(* IEC 61131-3 sources: RL_MAR/experiments/results/ablation/Ablation_no_post_process_deepseek-ai_DeepSeek-V3.2_20260602_235132 (part 2) *)

(* ---- med_34.st ---- *)
(*
    Coffee Machine Control Function Block
    Implements sequential control for water heating, grinding, and brewing
    Only one process active at a time
    Resets when start button is released
*)

FUNCTION_BLOCK CoffeeMachineControl
VAR_INPUT
    StartButton : BOOL;                    (* Start/run command *)
    ElapsedTime : DINT;                    (* Time elapsed since process start in ms *)
END_VAR

VAR_OUTPUT
    WaterHeating : BOOL;                   (* Control signal for water heater *)
    GrinderRunning : BOOL;                 (* Control signal for coffee grinder *)
    Brewing : BOOL;                        (* Control signal for brewing pump *)
    WaterHeated : BOOL;                    (* Status: Water heating complete *)
    GrinderFinished : BOOL;                (* Status: Grinding complete *)
    CoffeeReady : BOOL;                    (* Status: Brewing complete *)
END_VAR

VAR
    (* Process timing constants *)
    WaterHeatingDuration : DINT := 30000;  (* 30 seconds in milliseconds *)
    GrinderDuration : DINT := 15000;       (* 15 seconds in milliseconds *)
    BrewingDuration : DINT := 60000;       (* 60 seconds in milliseconds *)

    (* State management *)
    CurrentState : INT := 0;               (* 0=Idle, 1=Heating, 2=Grinding, 3=Brewing *)
    StateStartTime : DINT := 0;            (* Time when current state started *)
    PreviousStartButton : BOOL := FALSE;   (* Edge detection for start button *)

    (* Internal flags *)
    InternalWaterHeated : BOOL := FALSE;
    InternalGrinderFinished : BOOL := FALSE;
    InternalCoffeeReady : BOOL := FALSE;
END_VAR

(* Main control logic *)
IF NOT StartButton THEN
    (* Reset all outputs and state when start button is not pressed *)
    CurrentState := 0;
    StateStartTime := 0;
    WaterHeating := FALSE;
    GrinderRunning := FALSE;
    Brewing := FALSE;
    InternalWaterHeated := FALSE;
    InternalGrinderFinished := FALSE;
    InternalCoffeeReady := FALSE;
ELSE
    (* Detect rising edge of start button *)
    IF StartButton AND NOT PreviousStartButton AND CurrentState = 0 THEN
        (* Start new cycle from idle state *)
        CurrentState := 1;
        StateStartTime := ElapsedTime;
        InternalWaterHeated := FALSE;
        InternalGrinderFinished := FALSE;
        InternalCoffeeReady := FALSE;
    END_IF;

    (* State machine execution *)
    CASE CurrentState OF
        0: (* Idle State *)
            WaterHeating := FALSE;
            GrinderRunning := FALSE;
            Brewing := FALSE;

        1: (* Water Heating State *)
            WaterHeating := TRUE;
            GrinderRunning := FALSE;
            Brewing := FALSE;

            (* Check if heating duration completed *)
            IF (ElapsedTime - StateStartTime) >= WaterHeatingDuration THEN
                InternalWaterHeated := TRUE;
                WaterHeating := FALSE;
                CurrentState := 2;
                StateStartTime := ElapsedTime;
            END_IF;

        2: (* Grinding State *)
            WaterHeating := FALSE;
            GrinderRunning := TRUE;
            Brewing := FALSE;

            (* Check if grinding duration completed *)
            IF (ElapsedTime - StateStartTime) >= GrinderDuration THEN
                InternalGrinderFinished := TRUE;
                GrinderRunning := FALSE;
                CurrentState := 3;
                StateStartTime := ElapsedTime;
            END_IF;

        3: (* Brewing State *)
            WaterHeating := FALSE;
            GrinderRunning := FALSE;
            Brewing := TRUE;

            (* Check if brewing duration completed *)
            IF (ElapsedTime - StateStartTime) >= BrewingDuration THEN
                InternalCoffeeReady := TRUE;
                Brewing := FALSE;
                CurrentState := 0;  (* Return to idle after completion *)
            END_IF;
    END_CASE;
END_IF;

(* Update status outputs *)
WaterHeated := InternalWaterHeated;
GrinderFinished := InternalGrinderFinished;
CoffeeReady := InternalCoffeeReady;

(* Store previous start button state for edge detection *)
PreviousStartButton := StartButton;

END_FUNCTION_BLOCK;

(* ---- med_35.st ---- *)
FUNCTION_BLOCK FB_SimpleCalculation
VAR_INPUT
    INPUT_VAR1 : INT := 2;
    VAR2 : INT := 0;
END_VAR

VAR_OUTPUT
    OUTPUT_VAR1 : INT;
    OUTPUT_VAR2 : INT;
END_VAR

VAR
    i : INT; // Loop counter for multiplication loop
    COUNTER2 : INT := 0;
END_VAR

// Initialize outputs from inputs
OUTPUT_VAR1 := INPUT_VAR1;
OUTPUT_VAR2 := VAR2;

// First loop: Multiply OUTPUT_VAR1 by 2 for exactly 5 iterations
FOR i := 1 TO 5 DO
    OUTPUT_VAR1 := OUTPUT_VAR1 * 2;
END_FOR;

// Second loop: Increment OUTPUT_VAR2 by 1 for exactly 5 iterations
COUNTER2 := 0;
WHILE COUNTER2 < 5 DO
    OUTPUT_VAR2 := OUTPUT_VAR2 + 1;
    COUNTER2 := COUNTER2 + 1;
END_WHILE;

END_FUNCTION_BLOCK

(* ---- med_36.st ---- *)
TYPE
    Point2D : STRUCT
        X : INT;
        Y : INT;
    END_STRUCT;
END_TYPE

FUNCTION_BLOCK FB_ExpandedPoint
    VAR_INPUT
        INPUT_VAR2 : INT;
        INPUT_VAR1_X : INT;
        INPUT_VAR1_Y : INT;
        INPUT_VAR3_X : INT := 1;
        INPUT_VAR3_Y : INT := 2;
    END_VAR

    VAR_OUTPUT
        OUTPUT_VAR2 : INT;
        OUTPUT_VAR1_X : INT;
        OUTPUT_VAR1_Y : INT;
        OUTPUT_VAR3_X : INT;
        OUTPUT_VAR3_Y : INT;
    END_VAR

    VAR
        // Internal structured variables for cleaner code organization
        Internal_INPUT_VAR1 : Point2D;
        Internal_INPUT_VAR3 : Point2D;
        Internal_OUTPUT_VAR1 : Point2D;
        Internal_OUTPUT_VAR3 : Point2D;
    END_VAR

    // Main execution logic
    OUTPUT_VAR2 := INPUT_VAR2;

    // Set OUTPUT_VAR1_X and OUTPUT_VAR1_Y to fixed constants as specified
    OUTPUT_VAR1_X := 1;
    OUTPUT_VAR1_Y := 2;

    // Set OUTPUT_VAR3_X and OUTPUT_VAR3_Y to fixed constants as specified
    OUTPUT_VAR3_X := 100;
    OUTPUT_VAR3_Y := -7000;

    // Optional: Update internal structured variables for consistency
    Internal_OUTPUT_VAR1.X := OUTPUT_VAR1_X;
    Internal_OUTPUT_VAR1.Y := OUTPUT_VAR1_Y;
    Internal_OUTPUT_VAR3.X := OUTPUT_VAR3_X;
    Internal_OUTPUT_VAR3.Y := OUTPUT_VAR3_Y;

    // Store input values in internal structured variables (for potential future use)
    Internal_INPUT_VAR1.X := INPUT_VAR1_X;
    Internal_INPUT_VAR1.Y := INPUT_VAR1_Y;
    Internal_INPUT_VAR3.X := INPUT_VAR3_X;
    Internal_INPUT_VAR3.Y := INPUT_VAR3_Y;

END_FUNCTION_BLOCK

(* ---- med_37.st ---- *)
FUNCTION_BLOCK FB_RealValueAdjuster
VAR_INPUT
    x_in : REAL;
END_VAR

VAR_OUTPUT
    x_out : REAL;
END_VAR

VAR
    x_int : INT;
END_VAR

x_out := x_in;

IF x_in = 0.0 THEN
    x_out := x_out + 1.0;
END_IF;

IF x_in <> 0.0 THEN
    x_out := x_out + 1.0;
END_IF;

x_int := REAL_TO_INT(x_in);
IF x_int <> 0 THEN
    x_out := x_out + 1.0;
END_IF;

END_FUNCTION_BLOCK

(* ---- med_38.st ---- *)
FUNCTION_BLOCK SolarPanelTracking
VAR_INPUT
    SolarIntensity : REAL;      (* Input: Solar intensity in percentage *)
    CurrentTime : TIME;         (* Input: Current time of day *)
END_VAR

VAR_OUTPUT
    PanelAngle : REAL := 0.0;   (* Output: Panel angle in degrees *)
END_VAR

VAR
    SunriseTime : TIME := T#6H;    (* Sunrise time set to 6 AM *)
    SunsetTime : TIME := T#18H;    (* Sunset time set to 6 PM *)
    NoonTime : TIME := T#12H;      (* Noon time set to 12 PM *)
    MorningAngle : REAL := 30.0;   (* Angle during morning *)
    NoonAngle : REAL := 60.0;      (* Angle during noon *)
    EveningAngle : REAL := 30.0;   (* Angle during evening *)
    State : INT := 0;              (* Current state *)
    NextState : INT := 0;          (* Next state *)
END_VAR

(* State machine implementation *)
CASE State OF
    0: (* INIT *)
        PanelAngle := 0.0;
        NextState := 1;

    1: (* CHECK_TIME *)
        IF (CurrentTime < SunriseTime) OR (CurrentTime >= SunsetTime) THEN
            NextState := 2; (* NIGHT *)
        ELSIF (CurrentTime >= SunriseTime) AND (CurrentTime < NoonTime) THEN
            NextState := 3; (* MORNING *)
        ELSIF (CurrentTime >= NoonTime) AND (CurrentTime < SunsetTime) THEN
            NextState := 4; (* AFTERNOON *)
        ELSE
            NextState := 2; (* Default to NIGHT for safety *)
        END_IF;

    2: (* NIGHT *)
        PanelAngle := 0.0;
        IF (CurrentTime >= SunriseTime) AND (CurrentTime < SunsetTime) THEN
            NextState := 1; (* Return to CHECK_TIME *)
        ELSE
            NextState := 2; (* Stay in NIGHT *)
        END_IF;

    3: (* MORNING *)
        PanelAngle := MorningAngle;
        IF SolarIntensity >= 90.0 THEN
            NextState := 5; (* HIGH_INTENSITY *)
        ELSIF CurrentTime >= NoonTime THEN
            NextState := 1; (* Return to CHECK_TIME *)
        ELSE
            NextState := 3; (* Stay in MORNING *)
        END_IF;

    4: (* AFTERNOON *)
        PanelAngle := EveningAngle;
        IF SolarIntensity >= 90.0 THEN
            NextState := 5; (* HIGH_INTENSITY *)
        ELSIF (CurrentTime < NoonTime) OR (CurrentTime >= SunsetTime) THEN
            NextState := 1; (* Return to CHECK_TIME *)
        ELSE
            NextState := 4; (* Stay in AFTERNOON *)
        END_IF;

    5: (* HIGH_INTENSITY *)
        PanelAngle := NoonAngle;
        IF SolarIntensity < 90.0 THEN
            NextState := 1; (* Return to CHECK_TIME *)
        ELSIF (CurrentTime < SunriseTime) OR (CurrentTime >= SunsetTime) THEN
            NextState := 2; (* Transition to NIGHT *)
        ELSE
            NextState := 5; (* Stay in HIGH_INTENSITY *)
        END_IF;

    ELSE
        (* Invalid state - reset to INIT *)
        State := 0;
        NextState := 0;
END_CASE;

(* Update state for next execution cycle *)
State := NextState;

(* CRITICAL: Ensure panel angle stays within 0 to 90 degrees *)
(* This handles both internal parameter errors and any edge cases *)
IF PanelAngle < 0.0 THEN
    PanelAngle := 0.0;
ELSIF PanelAngle > 90.0 THEN
    PanelAngle := 90.0;
END_IF;

END_FUNCTION_BLOCK

(* ---- med_39.st ---- *)
FUNCTION_BLOCK WindTurbineControl
VAR_INPUT
    WindSpeedSensor : REAL; (* Input for measuring wind speed *)
    GeneratorSpeedSensor : REAL; (* Input for measuring generator speed *)
END_VAR

VAR_OUTPUT
    BladePitch : INT; (* Output for blade pitch control (degrees) *)
    GeneratorSpeed : REAL; (* Output for generator speed control (RPM) *)
END_VAR

VAR
    (* No internal variables required for this simple logic *)
END_VAR

(* Main control logic based on wind speed categories *)
IF WindSpeedSensor <= 3.0 THEN
    (* Low wind speed: optimize for starting torque *)
    BladePitch := -5;
    GeneratorSpeed := 500.0;
ELSIF (WindSpeedSensor > 3.0) AND (WindSpeedSensor <= 5.0) THEN
    (* Moderate wind speed: optimal power generation *)
    BladePitch := 0;
    GeneratorSpeed := 800.0;
ELSE
    (* High wind speed: limit power to protect turbine *)
    BladePitch := 5;
    GeneratorSpeed := 1000.0;
END_IF;

END_FUNCTION_BLOCK

(* ---- med_40.st ---- *)
FUNCTION_BLOCK RockClimbingWallControl
VAR_INPUT
    UserWeightSensor : REAL; (* Input for measuring the user's weight *)
    WallDifficultyLevel : INT; (* Input for setting the wall's initial difficulty level *)
    WallHeight : REAL; (* Input for setting the wall's height *)
    RouteSelector : INT; (* Input for selecting a climbing route *)
END_VAR
VAR_OUTPUT
    ClimbingMotorSpeed : REAL; (* Output for controlling the climbing wall motor speed *)
    WallLights : BOOL; (* Output for controlling wall lighting *)
END_VAR
VAR
    nCurrentDifficulty : INT;
    rSpeedMultiplier : REAL;
END_VAR

(* Determine motor speed multiplier based on user weight *)
IF UserWeightSensor > 60.0 THEN
    rSpeedMultiplier := 1.0;
ELSE
    rSpeedMultiplier := 0.8;
END_IF;

(* Determine current difficulty level based on route selection *)
CASE RouteSelector OF
    1: nCurrentDifficulty := 1;
    2: nCurrentDifficulty := 2;
    3: nCurrentDifficulty := 3;
    ELSE
        nCurrentDifficulty := WallDifficultyLevel;
END_CASE;

(* Calculate final motor speed: multiplier * (1.0 + 0.1*(difficulty-1)) *)
ClimbingMotorSpeed := rSpeedMultiplier * (1.0 + (0.1 * (nCurrentDifficulty - 1)));

(* Control wall lights based on wall height *)
IF WallHeight > 5.0 THEN
    WallLights := TRUE;
ELSE
    WallLights := FALSE;
END_IF;

END_FUNCTION_BLOCK

(* ---- med_41.st ---- *)
FUNCTION_BLOCK FishTankControl
VAR_INPUT
    OxygenLevel : REAL;        (* Input for oxygen level in the tank *)
    WaterTemperature : REAL;   (* Input for water temperature *)
    FeedingTime : TIME;        (* Time for scheduled feeding *)
    CurrentTime : TIME;        (* Current system time *)
END_VAR
VAR_OUTPUT
    OxygenValve : BOOL;        (* Output to control oxygen supply *)
    Heater : BOOL;             (* Output to control the heater *)
    Feeder : BOOL;             (* Output to control the fish feeder *)
END_VAR
VAR
    FeedingActive : BOOL;      (* Internal flag for feeding status *)
END_VAR

(* Oxygen Control Logic *)
IF OxygenLevel < 5.0 THEN
    OxygenValve := TRUE;
ELSE
    OxygenValve := FALSE;
END_IF;

(* Heater Control Logic *)
IF WaterTemperature < 25.0 THEN
    Heater := TRUE;
ELSE
    Heater := FALSE;
END_IF;

(* Feeder Control Logic *)
FeedingActive := (CurrentTime >= FeedingTime);
IF FeedingActive THEN
    Feeder := TRUE;
ELSE
    Feeder := FALSE;
END_IF;

END_FUNCTION_BLOCK

(* ---- med_42.st ---- *)
FUNCTION_BLOCK RetractableRoofControl
VAR_INPUT
    RainSensor : BOOL; (* Input to detect rain *)
    WindSensor : BOOL; (* Input to detect wind *)
    TemperatureSensor : REAL; (* Input to measure temperature *)
END_VAR
VAR_OUTPUT
    RoofMotor : BOOL; (* Output to control the roof motor *)
END_VAR
VAR
    (* No internal variables required for this logic *)
END_VAR

BEGIN
    IF RainSensor AND WindSensor THEN
        RoofMotor := FALSE; (* Close completely *)
    ELSIF RainSensor AND NOT WindSensor THEN
        RoofMotor := TRUE; (* Partially closed *)
    ELSIF NOT RainSensor AND TemperatureSensor < 20.0 THEN
        RoofMotor := TRUE; (* Close slightly *)
    ELSIF NOT RainSensor AND TemperatureSensor >= 20.0 THEN
        RoofMotor := FALSE; (* Fully open *)
    ELSE
        RoofMotor := FALSE; (* Default state - safety fallback *)
    END_IF;
END_FUNCTION_BLOCK

(* ---- med_43.st ---- *)
FUNCTION_BLOCK SandwichMaker
VAR_INPUT
    BreadFeeder : BOOL; (* Input: Detects the presence of bread slices *)
    Ingredient1 : BOOL; (* Input: Detects the presence of Ingredient 1 (e.g., cheese) *)
    Ingredient2 : BOOL; (* Input: Detects the presence of Ingredient 2 (e.g., lettuce) *)
    Ingredient3 : BOOL; (* Input: Detects the presence of Ingredient 3 (e.g., tomatoes) *)
    Condiment1 : BOOL; (* Input: Detects the presence of Condiment 1 (e.g., mayo) *)
    Condiment2 : BOOL; (* Input: Detects the presence of Condiment 2 (e.g., mustard) *)
END_VAR
VAR_OUTPUT
    ConveyorMotor : BOOL; (* Output: Controls the conveyor belt motor *)
    AssembleMotor : BOOL; (* Output: Controls the sandwich assembly motor *)
END_VAR
VAR
    SliceCount : INT := 0; (* Counter for bread slices *)
    PrevBreadState : BOOL := FALSE; (* Previous state for edge detection *)
    AllIngredientsPresent : BOOL; (* Flag for ingredient availability *)
END_VAR

(* Edge detection for bread slice counting *)
IF BreadFeeder AND NOT PrevBreadState THEN
    SliceCount := SliceCount + 1;
END_IF;

(* Update previous bread state for next cycle *)
PrevBreadState := BreadFeeder;

(* Calculate ingredient availability *)
AllIngredientsPresent := Ingredient1 AND Ingredient2 AND Ingredient3 AND Condiment1 AND Condiment2;

(* Control conveyor motor based on bread presence *)
ConveyorMotor := BreadFeeder AND NOT AssembleMotor; (* Interlock: conveyor stops during assembly *)

(* Control assembly motor based on conditions *)
IF (SliceCount >= 2) AND AllIngredientsPresent THEN
    AssembleMotor := TRUE;
    (* Reset slice count after successful assembly *)
    SliceCount := 0;
ELSE
    AssembleMotor := FALSE;
END_IF;

(* Safety interlock: reset slice count if ingredients missing during operation *)
IF NOT AllIngredientsPresent AND SliceCount > 0 THEN
    SliceCount := 0;
END_IF;

END_FUNCTION_BLOCK

(* ---- med_44.st ---- *)
(*
FUNCTION_BLOCK: DroneChargingStation
DESCRIPTION: Manages charging and deployment for three drones based on battery levels.
INPUTS:
    Drone1BatteryLevel, Drone2BatteryLevel, Drone3BatteryLevel: INT (0-100%)
    ChargingTime: TIME - Duration for a full charge cycle.
OUTPUTS:
    Drone1Status, Drone2Status, Drone3Status: BOOL - Active charging status.
    ChargingStationStatus: BOOL - Station busy indicator.
    DroneDeployed: BOOL - Global deployment status.
INTERNALS:
    Uses a TON timer for precise charging duration.
    Implements priority-based charging (Drone1 > Drone2 > Drone3) when battery < 20%.
    Recalls deployment (sets DroneDeployed FALSE) if any drone battery falls below 10%.
    Auto-deploys a drone (sets DroneDeployed TRUE) if battery >= 80% and station is idle.
*)

FUNCTION_BLOCK DroneChargingStation
VAR_INPUT
    Drone1BatteryLevel : INT := 0; (* Battery level of Drone 1 (0-100%) *)
    Drone2BatteryLevel : INT := 0; (* Battery level of Drone 2 (0-100%) *)
    Drone3BatteryLevel : INT := 0; (* Battery level of Drone 3 (0-100%) *)
    ChargingTime : TIME := T#30s; (* Required charging duration per drone *)
END_VAR
VAR_OUTPUT
    Drone1Status : BOOL := FALSE; (* TRUE if Drone 1 is currently charging *)
    Drone2Status : BOOL := FALSE; (* TRUE if Drone 2 is currently charging *)
    Drone3Status : BOOL := FALSE; (* TRUE if Drone 3 is currently charging *)
    ChargingStationStatus : BOOL := FALSE; (* TRUE if station is busy charging *)
    DroneDeployed : BOOL := FALSE; (* TRUE if a drone is currently deployed *)
END_VAR
VAR
    ChargingTimer : TON; (* Standard On-Delay Timer for charging *)
    CurrentDrone : INT := 0; (* 0=None, 1=Drone1, 2=Drone2, 3=Drone3 *)
    State : INT := 0; (* 0=Idle, 1=Charging Drone1, 2=Charging Drone2, 3=Charging Drone3 *)
    PrevState : INT := 0;
END_VAR

(* Main State Machine Logic *)
PrevState := State;

CASE State OF
    0: (* IDLE - Station Available *)
        (* Reset charging outputs *)
        Drone1Status := FALSE;
        Drone2Status := FALSE;
        Drone3Status := FALSE;
        ChargingStationStatus := FALSE;
        CurrentDrone := 0;
        ChargingTimer(IN:=FALSE); (* Ensure timer is reset *)

        (* Priority check for drones needing charge (Battery < 20%) *)
        (* Charging only starts if no drone is currently deployed *)
        IF NOT DroneDeployed THEN
            IF Drone1BatteryLevel < 20 THEN
                State := 1;
                CurrentDrone := 1;
            ELSIF Drone2BatteryLevel < 20 THEN
                State := 2;
                CurrentDrone := 2;
            ELSIF Drone3BatteryLevel < 20 THEN
                State := 3;
                CurrentDrone := 3;
            END_IF;
        END_IF;

    1: (* CHARGING DRONE 1 *)
        (* Set outputs for Drone 1 *)
        Drone1Status := TRUE;
        ChargingStationStatus := TRUE;

        (* Start the charging timer if just entered this state *)
        IF PrevState <> State THEN
            ChargingTimer(IN:=TRUE, PT:=ChargingTime);
        END_IF;

        (* Check for deployment recall condition (any battery < 10%) *)
        IF (Drone1BatteryLevel < 10) OR (Drone2BatteryLevel < 10) OR (Drone3BatteryLevel < 10) THEN
            DroneDeployed := FALSE;
        END_IF;

        (* Check if charging is complete *)
        ChargingTimer(IN:=TRUE, PT:=ChargingTime);
        IF ChargingTimer.Q THEN
            ChargingTimer(IN:=FALSE);
            State := 0; (* Return to IDLE *)
        END_IF;

    2: (* CHARGING DRONE 2 *)
        (* Set outputs for Drone 2 *)
        Drone2Status := TRUE;
        ChargingStationStatus := TRUE;

        (* Start the charging timer if just entered this state *)
        IF PrevState <> State THEN
            ChargingTimer(IN:=TRUE, PT:=ChargingTime);
        END_IF;

        (* Check for deployment recall condition (any battery < 10%) *)
        IF (Drone1BatteryLevel < 10) OR (Drone2BatteryLevel < 10) OR (Drone3BatteryLevel < 10) THEN
            DroneDeployed := FALSE;
        END_IF;

        (* Check if charging is complete *)
        ChargingTimer(IN:=TRUE, PT:=ChargingTime);
        IF ChargingTimer.Q THEN
            ChargingTimer(IN:=FALSE);
            State := 0; (* Return to IDLE *)
        END_IF;

    3: (* CHARGING DRONE 3 *)
        (* Set outputs for Drone 3 *)
        Drone3Status := TRUE;
        ChargingStationStatus := TRUE;

        (* Start the charging timer if just entered this state *)
        IF PrevState <> State THEN
            ChargingTimer(IN:=TRUE, PT:=ChargingTime);
        END_IF;

        (* Check for deployment recall condition (any battery < 10%) *)
        IF (Drone1BatteryLevel < 10) OR (Drone2BatteryLevel < 10) OR (Drone3BatteryLevel < 10) THEN
            DroneDeployed := FALSE;
        END_IF;

        (* Check if charging is complete *)
        ChargingTimer(IN:=TRUE, PT:=ChargingTime);
        IF ChargingTimer.Q THEN
            ChargingTimer(IN:=FALSE);
            State := 0; (* Return to IDLE *)
        END_IF;
END_CASE;

(* Auto-Deployment Logic *)
(* A drone can be auto-deployed if the station is idle, no drone is currently deployed, and its battery is sufficient (>= 80%). *)
(* This logic is evaluated independently of the charging state machine. *)
IF (State = 0) AND (NOT DroneDeployed) THEN
    IF (Drone1BatteryLevel >= 80) AND (CurrentDrone <> 1) THEN
        DroneDeployed := TRUE;
    ELSIF (Drone2BatteryLevel >= 80) AND (CurrentDrone <> 2) THEN
        DroneDeployed := TRUE;
    ELSIF (Drone3BatteryLevel >= 80) AND (CurrentDrone <> 3) THEN
        DroneDeployed := TRUE;
    END_IF;
END_IF;

END_FUNCTION_BLOCK

(* ---- med_45.st ---- *)
FUNCTION_BLOCK AutomatedSmoothieMaker
VAR_INPUT
    BananaAvailable : BOOL;
    BerryMixAvailable : BOOL;
    SpinachAvailable : BOOL;
    YogurtAvailable : BOOL;
    CustomerPreference : INT;
END_VAR

VAR_OUTPUT
    BlenderMotor : BOOL;
    Dispenser : BOOL;
END_VAR

VAR
    RecipeValid : BOOL;
    IngredientsAvailable : BOOL;
END_VAR

(* Initialize outputs to safe state *)
BlenderMotor := FALSE;
Dispenser := FALSE;

(* Reset internal flags *)
RecipeValid := FALSE;
IngredientsAvailable := FALSE;

(* Validate customer preference and check ingredient availability *)
CASE CustomerPreference OF
    1:
        RecipeValid := TRUE;
        IngredientsAvailable := BananaAvailable AND BerryMixAvailable AND YogurtAvailable;
    2:
        RecipeValid := TRUE;
        IngredientsAvailable := BerryMixAvailable AND SpinachAvailable AND YogurtAvailable;
    3:
        RecipeValid := TRUE;
        IngredientsAvailable := BananaAvailable AND SpinachAvailable AND YogurtAvailable;
    ELSE
        RecipeValid := FALSE;
        IngredientsAvailable := FALSE;
END_CASE;

(* Activate outputs only when recipe is valid AND all ingredients are available *)
IF RecipeValid AND IngredientsAvailable THEN
    Dispenser := TRUE;
    BlenderMotor := TRUE;
ELSE
    Dispenser := FALSE;
    BlenderMotor := FALSE;
END_IF;

END_FUNCTION_BLOCK

(* ---- med_46.st ---- *)
FUNCTION_BLOCK PrecisionEngravingMachine
VAR_INPUT
    DesignSelection : INT;
END_VAR

VAR_OUTPUT
    EngravingDepth : REAL;
    EngravingSpeed : REAL;
    ZAxisMotor : BOOL;
    EngravingMotor : BOOL;
END_VAR

VAR
    CalculatedDepth : REAL;
    CalculatedSpeed : REAL;
END_VAR

(* Main logic: Evaluate design selection and set parameters accordingly *)
CASE DesignSelection OF
    1:
        CalculatedSpeed := 10.0;
        CalculatedDepth := 0.1;
        ZAxisMotor := TRUE;
        EngravingMotor := TRUE;
    2:
        CalculatedSpeed := 8.0;
        CalculatedDepth := 0.2;
        ZAxisMotor := TRUE;
        EngravingMotor := TRUE;
    3:
        CalculatedSpeed := 12.0;
        CalculatedDepth := 0.15;
        ZAxisMotor := TRUE;
        EngravingMotor := TRUE;
ELSE
        (* Invalid design: Disable motors and zero parameters *)
        CalculatedSpeed := 0.0;
        CalculatedDepth := 0.0;
        ZAxisMotor := FALSE;
        EngravingMotor := FALSE;
END_CASE;

(* Map calculated values to outputs *)
EngravingSpeed := CalculatedSpeed;
EngravingDepth := CalculatedDepth;

END_FUNCTION_BLOCK

(* ---- med_47.st ---- *)
FUNCTION_BLOCK WindowCleaningSystem
VAR_INPUT
    StartButton : BOOL;
    EmergencyStop : BOOL;
    UpperLimit : BOOL;
    LowerLimit : BOOL;
END_VAR

VAR_OUTPUT
    ElevatorUp : BOOL;
    ElevatorDown : BOOL;
    RotateClockwise : BOOL;
    WaterPump : BOOL;
END_VAR

VAR
    CleaningInProgress : BOOL;
    AtUpperLimitLatch : BOOL;
    StartRisingEdge : R_TRIG;
END_VAR

(* Emergency Stop has absolute highest priority *)
IF EmergencyStop THEN
    CleaningInProgress := FALSE;
    AtUpperLimitLatch := FALSE;
    ElevatorUp := FALSE;
    ElevatorDown := FALSE;
    RotateClockwise := FALSE;
    WaterPump := FALSE;
    RETURN; (* Exit immediately to prevent any further logic execution *)
END_IF;

(* Detect rising edge of StartButton for safe initiation *)
StartRisingEdge(CLK := StartButton);

(* State transition logic *)
IF NOT CleaningInProgress THEN
    (* Idle state - waiting for valid start command *)
    IF StartRisingEdge.Q AND NOT UpperLimit AND LowerLimit THEN
        CleaningInProgress := TRUE;
        AtUpperLimitLatch := FALSE;
    END_IF;
ELSE
    (* Active cleaning cycle *)
    IF NOT AtUpperLimitLatch THEN
        (* Phase 1: Moving Up *)
        IF UpperLimit THEN
            AtUpperLimitLatch := TRUE;
        END_IF;
    ELSE
        (* Phase 2: Cleaning while Moving Down *)
        IF LowerLimit THEN
            CleaningInProgress := FALSE;
            AtUpperLimitLatch := FALSE;
        END_IF;
    END_IF;
END_IF;

(* Output logic with explicit mutual exclusion and safety interlocks *)
ElevatorUp := CleaningInProgress AND NOT AtUpperLimitLatch AND NOT UpperLimit;
ElevatorDown := CleaningInProgress AND AtUpperLimitLatch AND NOT LowerLimit;
RotateClockwise := CleaningInProgress AND AtUpperLimitLatch AND NOT LowerLimit;
WaterPump := CleaningInProgress AND AtUpperLimitLatch AND NOT LowerLimit;

(* Final safety override - ensure no conflicting outputs *)
IF ElevatorUp AND ElevatorDown THEN
    ElevatorUp := FALSE;
    ElevatorDown := FALSE;
END_IF;

END_FUNCTION_BLOCK;

(* ---- med_48.st ---- *)
FUNCTION_BLOCK ChargingStationControl
VAR_INPUT
    EVConnected : BOOL;
    EVVoltage : REAL;
    EVCurrent : REAL;
    EVStateOfCharge : REAL;
    ChargingTimer : TIME;
    MinimumVoltage : REAL;
    MaximumCurrent : REAL;
    MinimumSOC : REAL;
    ChargingVoltage : REAL;
    ChargingCurrent : REAL;
    MaximumChargingTime : TIME;
END_VAR

VAR_OUTPUT
    EVCharging : BOOL;
END_VAR

VAR
    bStartConditionsMet : BOOL;
    bStopConditionActive : BOOL;
END_VAR

(* Evaluate all start conditions simultaneously *)
bStartConditionsMet := EVConnected AND
                       (EVVoltage > MinimumVoltage) AND
                       (EVCurrent <= MaximumCurrent) AND
                       (EVStateOfCharge < 100.0) AND
                       (ChargingTimer <= MaximumChargingTime);

(* Evaluate stop conditions independently - any single condition triggers stop *)
bStopConditionActive := NOT EVConnected OR
                        (EVVoltage <= MinimumVoltage) OR
                        (EVCurrent > MaximumCurrent) OR
                        (EVStateOfCharge >= 100.0) OR
                        (ChargingTimer > MaximumChargingTime);

(* Control logic: Start charging only when all start conditions are met AND no stop conditions are active *)
IF bStartConditionsMet AND NOT bStopConditionActive THEN
    EVCharging := TRUE;
ELSE
    EVCharging := FALSE;
END_IF;

END_FUNCTION_BLOCK;

(* ---- med_49.st ---- *)
TYPE
    // System status enumeration
    HVAC_SystemStatus : (
        STATUS_OFF := 0,
        STATUS_STANDBY,
        STATUS_HEATING,
        STATUS_COOLING,
        STATUS_VENTILATING,
        STATUS_FAULT
    );

    // Alarm status bits
    HVAC_AlarmBits : STRUCT
        TemperatureSensorFault : BOOL;
        HumiditySensorFault : BOOL;
        HeatingFault : BOOL;
        CoolingFault : BOOL;
        VentilationFault : BOOL;
        MaintenanceRequired : BOOL;
        _reserved : ARRAY[0..8] OF BOOL;
    END_STRUCT;
END_TYPE

FUNCTION_BLOCK SmartHVACSystem
VAR_INPUT
    // Primary sensor inputs
    TemperatureSensor : REAL; (* Raw temperature reading in °C *)
    HumiditySensor : REAL; (* Raw humidity reading in % *)

    // Configuration inputs
    DesiredTemperature : REAL := 24.0; (* Temperature setpoint *)
    DesiredHumidity : REAL := 50.0; (* Humidity setpoint *)
    TemperatureThreshold : REAL := 1.0; (* Temperature deadband *)
    HumidityThreshold : REAL := 5.0; (* Humidity deadband *)

    // Calibration inputs
    TemperatureCalibrationOffset : REAL := 0.0; (* Temperature calibration *)
    HumidityCalibrationOffset : REAL := 0.0; (* Humidity calibration *)

    // Control inputs
    ManualOverride : BOOL := FALSE; (* Manual override active *)
    ModeOverride : INT := 0; (* Manual mode: 0=Off, 1=Cooling, 2=Heating, 3=Ventilation *)
    FanSpeedOverride : INT := 0; (* Manual fan speed *)
    EmergencyStop : BOOL := FALSE; (* Emergency stop command *)

    // Hysteresis configuration
    TemperatureHysteresis : REAL := 0.5; (* Prevents rapid mode switching *)
    HumidityHysteresis : REAL := 2.0; (* Prevents rapid ventilation cycling *)

    // Timing configuration
    ModeChangeDelayTime : TIME := T#2s; (* Minimum time between mode changes *)
    SensorFilterTime : TIME := T#5s; (* Sensor filtering time constant *)
END_VAR

VAR_OUTPUT
    // Control outputs
    HVACMode : INT := 0; (* 0=Off, 1=Cooling, 2=Heating, 3=Ventilation *)
    HVACFanSpeed : INT := 0; (* 0=Off, 1=Low, 2=Medium, 3=High *)
    HeatingElement : BOOL := FALSE; (* Direct heating control *)
    CoolingCompressor : BOOL := FALSE; (* Direct cooling control *)
    VentilationDamper : REAL := 0.0; (* Ventilation damper position 0.0-100.0% *)

    // Status outputs
    SystemStatus : HVAC_SystemStatus := STATUS_OFF;
    TemperatureAlarm : BOOL := FALSE;
    HumidityAlarm : BOOL := FALSE;
    SystemAlarms : HVAC_AlarmBits;

    // Monitoring outputs
    EnergyConsumption : REAL := 0.0; (* Estimated energy consumption in kWh *)
    MaintenanceRequired : BOOL := FALSE;

    // Diagnostic outputs
    FilteredTemperature : REAL := 0.0;
    FilteredHumidity : REAL := 0.0;
    TemperatureError : REAL := 0.0;
    HumidityError : REAL := 0.0;
END_VAR

VAR
    // Sanitized and filtered values
    AdjustedTemperature : REAL;
    AdjustedHumidity : REAL;
    TemperatureFiltered : REAL;
    HumidityFiltered : REAL;

    // Requirement flags with hysteresis
    NeedsHeating : BOOL;
    NeedsCooling : BOOL;
    NeedsVentilationHigh : BOOL; (* For high humidity *)
    NeedsVentilationLow : BOOL; (* For low humidity *)

    // Hysteresis states
    HeatingHysteresisState : BOOL := FALSE;
    CoolingHysteresisState : BOOL := FALSE;
    VentilationHighHysteresisState : BOOL := FALSE;
    VentilationLowHysteresisState : BOOL := FALSE;

    // Control logic
    ActiveMode : INT := 0;
    ActiveFanSpeed : INT := 0;

    // Timing and delays
    ModeChangeDelay : TON;
    SensorFilterTimer : TON;

    // Counters and accumulators
    OperatingHoursCounter : DINT := 0;
    EnergyAccumulator : REAL := 0.0;
    MaintenanceCounter : DINT := 0;

    // State management
    PreviousMode : INT := 0;
    SystemState : INT := 0;

    // Internal calculations
    TemperatureCalibrated : REAL;
    HumidityCalibrated : REAL;
    EffectiveDesiredTemperature : REAL;
    EffectiveDesiredHumidity : REAL;

    // Fan speed calculation
    TemperatureDeviation : REAL;
    HumidityDeviation : REAL;
    CalculatedFanSpeed : INT;

    // Constants
    MIN_TEMPERATURE : REAL := -50.0;
    MAX_TEMPERATURE : REAL := 100.0;
    MIN_HUMIDITY : REAL := 0.0;
    MAX_HUMIDITY : REAL := 100.0;
    MAINTENANCE_INTERVAL : DINT := 8760; (* Hours between maintenance *)
END_VAR

// Main execution logic
// 1. Input sanitization and calibration
TemperatureCalibrated := TemperatureSensor + TemperatureCalibrationOffset;
HumidityCalibrated := HumiditySensor + HumidityCalibrationOffset;

// Sanitize temperature
IF TemperatureCalibrated < MIN_TEMPERATURE THEN
    AdjustedTemperature := MIN_TEMPERATURE;
    SystemAlarms.TemperatureSensorFault := TRUE;
ELSIF TemperatureCalibrated > MAX_TEMPERATURE THEN
    AdjustedTemperature := MAX_TEMPERATURE;
    SystemAlarms.TemperatureSensorFault := TRUE;
ELSE
    AdjustedTemperature := TemperatureCalibrated;
    SystemAlarms.TemperatureSensorFault := FALSE;
END_IF;

// Sanitize humidity
IF HumidityCalibrated < MIN_HUMIDITY THEN
    AdjustedHumidity := MIN_HUMIDITY;
    SystemAlarms.HumiditySensorFault := TRUE;
ELSIF HumidityCalibrated > MAX_HUMIDITY THEN
    AdjustedHumidity := MAX_HUMIDITY;
    SystemAlarms.HumiditySensorFault := TRUE;
ELSE
    AdjustedHumidity := HumidityCalibrated;
    SystemAlarms.HumiditySensorFault := FALSE;
END_IF;

// 2. Sensor filtering (simple moving average)
SensorFilterTimer(IN := NOT SensorFilterTimer.Q, PT := SensorFilterTime);
IF SensorFilterTimer.Q THEN
    TemperatureFiltered := (TemperatureFiltered * 0.9) + (AdjustedTemperature * 0.1);
    HumidityFiltered := (HumidityFiltered * 0.9) + (AdjustedHumidity * 0.1);
    SensorFilterTimer(IN := FALSE);
END_IF;

// 3. Calculate effective setpoints
EffectiveDesiredTemperature := DesiredTemperature;
EffectiveDesiredHumidity := DesiredHumidity;

// 4. Calculate errors
TemperatureError := EffectiveDesiredTemperature - TemperatureFiltered;
HumidityError := EffectiveDesiredHumidity - HumidityFiltered;

// 5. Determine requirements with hysteresis
// Heating requirement with hysteresis
IF TemperatureFiltered < (EffectiveDesiredTemperature - TemperatureThreshold) THEN
    NeedsHeating := TRUE;
    HeatingHysteresisState := TRUE;
ELSIF TemperatureFiltered > (EffectiveDesiredTemperature - TemperatureThreshold + TemperatureHysteresis) AND HeatingHysteresisState THEN
    NeedsHeating := FALSE;
    HeatingHysteresisState := FALSE;
END_IF;

// Cooling requirement with hysteresis
IF TemperatureFiltered > (EffectiveDesiredTemperature + TemperatureThreshold) THEN
    NeedsCooling := TRUE;
    CoolingHysteresisState := TRUE;
ELSIF TemperatureFiltered < (EffectiveDesiredTemperature + TemperatureThreshold - TemperatureHysteresis) AND CoolingHysteresisState THEN
    NeedsCooling := FALSE;
    CoolingHysteresisState := FALSE;
END_IF;

// Ventilation for high humidity with hysteresis
IF HumidityFiltered > (EffectiveDesiredHumidity + HumidityThreshold) THEN
    NeedsVentilationHigh := TRUE;
    VentilationHighHysteresisState := TRUE;
ELSIF HumidityFiltered < (EffectiveDesiredHumidity + HumidityThreshold - HumidityHysteresis) AND VentilationHighHysteresisState THEN
    NeedsVentilationHigh := FALSE;
    VentilationHighHysteresisState := FALSE;
END_IF;

// Ventilation for low humidity with hysteresis
IF HumidityFiltered < (EffectiveDesiredHumidity - HumidityThreshold) THEN
    NeedsVentilationLow := TRUE;
    VentilationLowHysteresisState := TRUE;
ELSIF HumidityFiltered > (EffectiveDesiredHumidity - HumidityThreshold + HumidityHysteresis) AND VentilationLowHysteresisState THEN
    NeedsVentilationLow := FALSE;
    VentilationLowHysteresisState := FALSE;
END_IF;

// 6. Mode selection with prioritization and mutual exclusion
ModeChangeDelay(IN := (ActiveMode <> PreviousMode), PT := ModeChangeDelayTime);

IF EmergencyStop THEN
    ActiveMode := 0;
    ActiveFanSpeed := 0;
    SystemStatus := STATUS_OFF;

ELSIF ManualOverride THEN
    ActiveMode := LIMIT(0, ModeOverride, 3);
    ActiveFanSpeed := LIMIT(0, FanSpeedOverride, 3);
    SystemStatus := HVAC_SystemStatus(ActiveMode + 1); // Map to status enum

ELSE
    // Normal automatic control with prioritization
    IF NeedsHeating AND NOT NeedsCooling THEN
        // Heating has priority
        IF ModeChangeDelay.Q OR ActiveMode = 2 THEN
            ActiveMode := 2; // Heating
            SystemStatus := STATUS_HEATING;
        END_IF;

    ELSIF NeedsCooling AND NOT NeedsHeating THEN
        // Cooling has priority (mutually exclusive with heating)
        IF ModeChangeDelay.Q OR ActiveMode = 1 THEN
            ActiveMode := 1; // Cooling
            SystemStatus := STATUS_COOLING;
        END_IF;

    ELSIF (NeedsVentilationHigh OR NeedsVentilationLow) AND NOT (NeedsHeating OR NeedsCooling) THEN
        // Ventilation only when no temperature control needed
        IF ModeChangeDelay.Q OR ActiveMode = 3 THEN
            ActiveMode := 3; // Ventilation
            SystemStatus := STATUS_VENTILATING;
        END_IF;

    ELSE
        // No requirements met
        ActiveMode := 0; // Off
        SystemStatus := STATUS_STANDBY;
    END_IF;

    // Calculate appropriate fan speed based on deviation
    TemperatureDeviation := ABS(TemperatureError);
    HumidityDeviation := ABS(HumidityError);

    CASE ActiveMode OF
        1, 2: // Heating or Cooling
            IF TemperatureDeviation > (TemperatureThreshold * 2) THEN
                CalculatedFanSpeed := 3; // High
            ELSIF TemperatureDeviation > TemperatureThreshold THEN
                CalculatedFanSpeed := 2; // Medium
            ELSE
                CalculatedFanSpeed := 1; // Low
            END_IF;

        3: // Ventilation
            IF HumidityDeviation > (HumidityThreshold * 2) THEN
                CalculatedFanSpeed := 3; // High
            ELSIF HumidityDeviation > HumidityThreshold THEN
                CalculatedFanSpeed := 2; // Medium
            ELSE
                CalculatedFanSpeed := 1; // Low
            END_IF;

        ELSE: // Off
            CalculatedFanSpeed := 0;
    END_CASE;

    ActiveFanSpeed := CalculatedFanSpeed;
END_IF;

// 7. Set direct control outputs with safety interlocks
HeatingElement := (ActiveMode = 2) AND NOT EmergencyStop AND NOT SystemAlarms.HeatingFault;
CoolingCompressor := (ActiveMode = 1) AND NOT EmergencyStop AND NOT SystemAlarms.CoolingFault;

// Ventilation damper position based on humidity error
IF ActiveMode = 3 THEN
    VentilationDamper := LIMIT(0.0, ABS(HumidityError) * 2.0, 100.0);
ELSE
    VentilationDamper := 0.0;
END_IF;

// 8. Update output variables
HVACMode := ActiveMode;
HVACFanSpeed := ActiveFanSpeed;

// 9. Update diagnostic outputs
FilteredTemperature := TemperatureFiltered;
FilteredHumidity := HumidityFiltered;

// 10. Alarm generation
TemperatureAlarm := SystemAlarms.TemperatureSensorFault OR (ABS(TemperatureError) > (TemperatureThreshold * 3));
HumidityAlarm := SystemAlarms.HumiditySensorFault OR (ABS(HumidityError) > (HumidityThreshold * 3));

// 11. Energy and maintenance tracking
IF ActiveMode <> 0 THEN
    OperatingHoursCounter := OperatingHoursCounter + 1;

    // Simple energy estimation
    CASE ActiveMode OF
        1: EnergyAccumulator := EnergyAccumulator + 3.5; // Cooling energy
        2: EnergyAccumulator := EnergyAccumulator + 4.0; // Heating energy
        3: EnergyAccumulator := EnergyAccumulator + 0.5; // Ventilation energy
    END_CASE;
END_IF;

EnergyConsumption := EnergyAccumulator;

// Maintenance tracking
MaintenanceCounter := OperatingHoursCounter;
MaintenanceRequired := (MaintenanceCounter >= MAINTENANCE_INTERVAL);
SystemAlarms.MaintenanceRequired := MaintenanceRequired;

// 12. Update previous mode for change detection
IF ModeChangeDelay.Q THEN
    PreviousMode := ActiveMode;
END_IF;

// 13. Fault status handling
IF EmergencyStop THEN
    SystemStatus := STATUS_OFF;
ELSIF SystemAlarms.TemperatureSensorFault OR SystemAlarms.HumiditySensorFault OR
      SystemAlarms.HeatingFault OR SystemAlarms.CoolingFault OR SystemAlarms.VentilationFault THEN
    SystemStatus := STATUS_FAULT;
END_IF;
END_FUNCTION_BLOCK;

(* ---- med_50.st ---- *)
TYPE
    // Define a FIFO queue structure for up to 50 pending requests per elevator
    ElevatorQueue : STRUCT
        Buffer : ARRAY[1..50] OF INT;
        Head : INT; // Points to the next element to be removed
        Tail : INT; // Points to the next free position for insertion
        Count : INT; // Number of elements currently in the queue
    END_STRUCT;
END_TYPE

FUNCTION_BLOCK CarParkingSystem
VAR_INPUT
    NewCarSlot : INT; (* Input for new car arrival slot number (1-100) *)
END_VAR
VAR_OUTPUT
    Elevator1Busy : BOOL; (* Elevator 1 status - TRUE when moving to target *)
    Elevator2Busy : BOOL; (* Elevator 2 status - TRUE when moving to target *)
    Elevator1Position : INT; (* Elevator 1 current position (1-50) *)
    Elevator2Position : INT; (* Elevator 2 current position (51-100) *)
END_VAR
VAR
    // Target positions for each elevator
    Elevator1Target : INT;
    Elevator2Target : INT;

    // Parking slot occupancy tracking (TRUE = occupied)
    CarSlots : ARRAY[1..100] OF BOOL;

    // Queues for pending requests when elevators are busy
    Queue1 : ElevatorQueue;
    Queue2 : ElevatorQueue;

    // Internal helper variables
    bInitComplete : BOOL := FALSE;
    iScanSlot : INT;
END_VAR

// ============================================================================
// INITIALIZATION - Executes once on first scan
// ============================================================================
IF NOT bInitComplete THEN
    // Initialize parking slots as empty
    FOR iScanSlot := 1 TO 100 DO
        CarSlots[iScanSlot] := FALSE;
    END_FOR;

    // Set initial elevator positions (home positions)
    Elevator1Position := 1;
    Elevator2Position := 51;
    Elevator1Target := 1;
    Elevator2Target := 51;

    // Set elevators to idle state
    Elevator1Busy := FALSE;
    Elevator2Busy := FALSE;

    // Initialize queues
    Queue1.Head := 1;
    Queue1.Tail := 1;
    Queue1.Count := 0;

    Queue2.Head := 1;
    Queue2.Tail := 1;
    Queue2.Count := 0;

    bInitComplete := TRUE;
END_IF;

// ============================================================================
// QUEUE MANAGEMENT FUNCTIONS (Local implementations)
// ============================================================================

// Function to add a slot to a queue (returns TRUE if successful)
IF (NewCarSlot >= 1) AND (NewCarSlot <= 100) AND (NOT CarSlots[NewCarSlot]) THEN
    CarSlots[NewCarSlot] := TRUE;

    CASE NewCarSlot OF
        1..50:
            // Assign to Elevator 1 zone
            IF NOT Elevator1Busy THEN
                // Elevator 1 is idle - assign directly
                Elevator1Target := NewCarSlot;
                Elevator1Busy := TRUE;
            ELSE
                // Elevator 1 is busy - add to queue if space available
                IF Queue1.Count < 50 THEN
                    Queue1.Buffer[Queue1.Tail] := NewCarSlot;
                    Queue1.Tail := Queue1.Tail + 1;
                    Queue1.Count := Queue1.Count + 1;

                    // Wrap tail pointer if necessary
                    IF Queue1.Tail > 50 THEN
                        Queue1.Tail := 1;
                    END_IF;
                END_IF;
                // If queue is full (50 pending requests), the arrival is ignored
            END_IF;

        51..100:
            // Assign to Elevator 2 zone
            IF NOT Elevator2Busy THEN
                // Elevator 2 is idle - assign directly
                Elevator2Target := NewCarSlot;
                Elevator2Busy := TRUE;
            ELSE
                // Elevator 2 is busy - add to queue if space available
                IF Queue2.Count < 50 THEN
                    Queue2.Buffer[Queue2.Tail] := NewCarSlot;
                    Queue2.Tail := Queue2.Tail + 1;
                    Queue2.Count := Queue2.Count + 1;

                    // Wrap tail pointer if necessary
                    IF Queue2.Tail > 50 THEN
                        Queue2.Tail := 1;
                    END_IF;
                END_IF;
                // If queue is full (50 pending requests), the arrival is ignored
            END_IF;
    END_CASE;
END_IF;

// ============================================================================
// ELEVATOR 1 MOTION CONTROL
// ============================================================================
IF Elevator1Busy THEN
    // Move elevator toward target (one slot per scan cycle)
    IF Elevator1Position < Elevator1Target THEN
        Elevator1Position := Elevator1Position + 1;
    ELSIF Elevator1Position > Elevator1Target THEN
        Elevator1Position := Elevator1Position - 1;
    ELSE
        // Reached target - elevator becomes idle
        Elevator1Busy := FALSE;

        // Check if there are pending requests in queue
        IF Queue1.Count > 0 THEN
            // Get next target from queue (FIFO)
            Elevator1Target := Queue1.Buffer[Queue1.Head];
            Queue1.Head := Queue1.Head + 1;
            Queue1.Count := Queue1.Count - 1;

            // Wrap head pointer if necessary
            IF Queue1.Head > 50 THEN
                Queue1.Head := 1;
            END_IF;

            // Elevator becomes busy again with new target
            Elevator1Busy := TRUE;
        END_IF;
    END_IF;
END_IF;

// ============================================================================
// ELEVATOR 2 MOTION CONTROL
// ============================================================================
IF Elevator2Busy THEN
    // Move elevator toward target (one slot per scan cycle)
    IF Elevator2Position < Elevator2Target THEN
        Elevator2Position := Elevator2Position + 1;
    ELSIF Elevator2Position > Elevator2Target THEN
        Elevator2Position := Elevator2Position - 1;
    ELSE
        // Reached target - elevator becomes idle
        Elevator2Busy := FALSE;

        // Check if there are pending requests in queue
        IF Queue2.Count > 0 THEN
            // Get next target from queue (FIFO)
            Elevator2Target := Queue2.Buffer[Queue2.Head];
            Queue2.Head := Queue2.Head + 1;
            Queue2.Count := Queue2.Count - 1;

            // Wrap head pointer if necessary
            IF Queue2.Head > 50 THEN
                Queue2.Head := 1;
            END_IF;

            // Elevator becomes busy again with new target
            Elevator2Busy := TRUE;
        END_IF;
    END_IF;
END_IF;

// ============================================================================
// IDLE ELEVATOR SCANNING
// ============================================================================
// Elevator 1 scans its zone (slots 1-50) when idle
IF NOT Elevator1Busy THEN
    FOR iScanSlot := 1 TO 50 DO
        IF CarSlots[iScanSlot] THEN
            // Found an occupied slot in zone - assign as target
            Elevator1Target := iScanSlot;
            Elevator1Busy := TRUE;
            EXIT; // Stop scanning after first assignment
        END_IF;
    END_FOR;
END_IF;

// Elevator 2 scans its zone (slots 51-100) when idle
IF NOT Elevator2Busy THEN
    FOR iScanSlot := 51 TO 100 DO
        IF CarSlots[iScanSlot] THEN
            // Found an occupied slot in zone - assign as target
            Elevator2Target := iScanSlot;
            Elevator2Busy := TRUE;
            EXIT; // Stop scanning after first assignment
        END_IF;
    END_FOR;
END_IF;

END_FUNCTION_BLOCK;

(* ---- med_51.st ---- *)
(*
FUNCTION_BLOCK: PizzaMakingMachine
DESCRIPTION: Oversees complete pizza production process with sequential control and safety interlocks.
AUTHOR: Senior PLC Commissioning Engineer
COMPLIANCE: IEC 61131-3 Structured Text
*)

FUNCTION_BLOCK PizzaMakingMachine
VAR_INPUT
    StartButton : BOOL;          (* Momentary start command *)
    StopButton : BOOL;           (* Emergency stop - stops all operations *)
    DoughReadySensor : BOOL;     (* TRUE when dough preparation complete *)
    ToppingsReadySensor : BOOL;  (* TRUE when toppings application complete *)
    BakingDoneSensor : BOOL;     (* TRUE when baking cycle complete *)
END_VAR

VAR_OUTPUT
    DoughRollerMotor : BOOL;     (* Controls dough roller mechanism *)
    ToppingDispenser : BOOL;     (* Controls topping application system *)
    ConveyorMotor : BOOL;        (* Controls pizza transfer to oven *)
    OvenHeater : BOOL;           (* Controls oven heating element *)
    OvenTemperature : INT;       (* Current oven temperature setpoint *)
END_VAR

VAR
    (* State Management *)
    MachineActive : BOOL;        (* Master enable for all operations *)
    BakingActive : BOOL;         (* Baking process active flag *)

    (* Timing Control *)
    BakeTimer : TON;             (* Baking duration timer *)
    BakeDuration : TIME := T#30S; (* Fixed 30-second baking time *)

    (* Safety Flags *)
    SafeToStart : BOOL;          (* System ready for start command *)
END_VAR

(*
MAIN LOGIC SEQUENCE:
1. Start/Stop Logic with safety interlocks
2. Dough Preparation Phase
3. Topping Application Phase
4. Transfer & Baking Phase
5. Temperature Control
6. Emergency Stop Override
*)

(* --- SAFETY AND START/STOP CONTROL --- *)
(* Stop button has priority - immediately disables all operations *)
IF StopButton THEN
    MachineActive := FALSE;
ELSIF StartButton AND NOT MachineActive THEN
    (* Allow start only when system is stopped and start button is pressed *)
    MachineActive := TRUE;
END_IF;

(* --- MAIN OPERATIONAL SEQUENCE --- *)
IF MachineActive THEN
    (* PHASE 1: DOUGH PREPARATION *)
    IF NOT DoughReadySensor THEN
        DoughRollerMotor := TRUE;
        ToppingDispenser := FALSE;
        ConveyorMotor := FALSE;
        BakingActive := FALSE;

    (* PHASE 2: TOPPING APPLICATION *)
    ELSIF DoughReadySensor AND NOT ToppingsReadySensor THEN
        DoughRollerMotor := FALSE;
        ToppingDispenser := TRUE;
        ConveyorMotor := FALSE;
        BakingActive := FALSE;

    (* PHASE 3: TRANSFER TO OVEN & BAKING *)
    ELSIF DoughReadySensor AND ToppingsReadySensor AND NOT BakingActive THEN
        DoughRollerMotor := FALSE;
        ToppingDispenser := FALSE;
        ConveyorMotor := TRUE;
        OvenHeater := TRUE;
        BakingActive := TRUE;

        (* Start baking timer when pizza enters oven *)
        BakeTimer(IN := TRUE, PT := BakeDuration);

    (* PHASE 4: BAKING IN PROGRESS *)
    ELSIF BakingActive THEN
        DoughRollerMotor := FALSE;
        ToppingDispenser := FALSE;
        ConveyorMotor := FALSE;  (* Conveyor stops during baking *)
        OvenHeater := TRUE;

        (* Continue timing the baking process *)
        BakeTimer(IN := TRUE, PT := BakeDuration);

        (* Check for baking completion - either by timer OR sensor *)
        IF BakeTimer.Q OR BakingDoneSensor THEN
            BakingActive := FALSE;
            OvenHeater := FALSE;
            BakeTimer(IN := FALSE);  (* Reset timer *)
        END_IF;
    END_IF;

    (* --- TEMPERATURE CONTROL --- *)
    IF OvenHeater THEN
        OvenTemperature := 220;  (* Baking temperature setpoint *)
    ELSE
        OvenTemperature := 0;    (* Oven off temperature *)
    END_IF;

ELSE
    (* --- EMERGENCY STOP / SYSTEM IDLE STATE --- *)
    DoughRollerMotor := FALSE;
    ToppingDispenser := FALSE;
    ConveyorMotor := FALSE;
    OvenHeater := FALSE;
    OvenTemperature := 0;
    BakingActive := FALSE;
    BakeTimer(IN := FALSE);  (* Ensure timer is reset *)
END_IF;

END_FUNCTION_BLOCK

(* ---- med_52.st ---- *)
FUNCTION_BLOCK TrafficManagementSystem
VAR_INPUT
    VehicleCount1 : INT;
    VehicleCount2 : INT;
    VehicleCount3 : INT;
    VehicleCount4 : INT;
END_VAR

VAR_OUTPUT
    TrafficLight1 : BOOL;
    TrafficLight2 : BOOL;
    TrafficLight3 : BOOL;
    TrafficLight4 : BOOL;
END_VAR

VAR
    // No internal variables needed for this implementation
END_VAR

// Pair 1: Intersection 1 vs Intersection 2
IF VehicleCount1 > VehicleCount2 THEN
    TrafficLight1 := TRUE;   // Green for intersection with higher count
    TrafficLight2 := FALSE;  // Red for the other intersection
ELSIF VehicleCount2 > VehicleCount1 THEN
    TrafficLight1 := FALSE;  // Red for intersection with lower count
    TrafficLight2 := TRUE;   // Green for the other intersection
ELSE
    // Equal counts: default priority to Intersection 1
    TrafficLight1 := TRUE;   // Green for Intersection 1
    TrafficLight2 := FALSE;  // Red for Intersection 2
END_IF;

// Pair 2: Intersection 3 vs Intersection 4
IF VehicleCount3 > VehicleCount4 THEN
    TrafficLight3 := TRUE;   // Green for intersection with higher count
    TrafficLight4 := FALSE;  // Red for the other intersection
ELSIF VehicleCount4 > VehicleCount3 THEN
    TrafficLight3 := FALSE;  // Red for intersection with lower count
    TrafficLight4 := TRUE;   // Green for the other intersection
ELSE
    // Equal counts: default priority to Intersection 3
    TrafficLight3 := TRUE;   // Green for Intersection 3
    TrafficLight4 := FALSE;  // Red for Intersection 4
END_IF;

END_FUNCTION_BLOCK

(* ---- med_53.st ---- *)
(*
    FUNCTION_BLOCK: PouchMachine
    Description: Controls the startup and shutdown sequences for a 3D pouch making machine.
    The machine includes 8 heating stations, 8 cooling stations, two feeder units,
    and one horizontal and one vertical cutter.
    Startup Sequence: Heating -> Cooling -> Feeders (with tension) -> Horizontal Cutter -> Vertical Cutter -> Ready.
    Shutdown Sequence: Cutters -> Feeders -> Heating -> Cooling -> Idle.
    The state machine can be interrupted at any time by the stop command.
*)

FUNCTION_BLOCK PouchMachine
VAR_INPUT
    start_machine: BOOL;    (* Rising edge triggers startup sequence from Idle *)
    stop_machine: BOOL;     (* Command to initiate shutdown sequence from any state *)
END_VAR

VAR_OUTPUT
    machine_ready: BOOL;    (* TRUE when machine is fully operational *)
    feeder_running: BOOL;   (* TRUE when both feeder units are running with tension *)
    cutter_running: BOOL;   (* TRUE when both horizontal and vertical cutters are active *)
    heating_running: BOOL;  (* TRUE when all 8 heating stations are active *)
    cooling_running: BOOL;  (* TRUE when all 8 cooling stations are active *)
END_VAR

VAR
    startup_complete: BOOL := FALSE;
    shutdown_complete: BOOL := FALSE;
    current_state: INT := 0;
    next_state: INT := 0;
END_VAR

(* Main State Machine Logic *)
CASE current_state OF
    0: (* Idle State - Machine is stopped and outputs are reset *)
        machine_ready := FALSE;
        feeder_running := FALSE;
        cutter_running := FALSE;
        heating_running := FALSE;
        cooling_running := FALSE;
        startup_complete := FALSE;
        shutdown_complete := FALSE;

        IF start_machine AND NOT stop_machine THEN
            next_state := 1; (* Begin startup sequence *)
        ELSE
            next_state := 0; (* Remain idle *)
        END_IF;

    1: (* Startup - Activate Heating Stations *)
        heating_running := TRUE; (* Activate all 8 heating stations *)

        IF heating_running AND NOT stop_machine THEN
            next_state := 2; (* Proceed to activate cooling *)
        ELSIF stop_machine THEN
            next_state := 6; (* Abort startup, begin shutdown *)
        ELSE
            next_state := 1; (* Wait for heating to be confirmed active *)
        END_IF;

    2: (* Startup - Activate Cooling Stations *)
        cooling_running := TRUE; (* Activate all 8 cooling stations *)

        IF cooling_running AND NOT stop_machine THEN
            next_state := 3; (* Proceed to start feeders *)
        ELSIF stop_machine THEN
            next_state := 6; (* Abort startup, begin shutdown *)
        ELSE
            next_state := 2; (* Wait for cooling to be confirmed active *)
        END_IF;

    3: (* Startup - Start Feeders with Tension Control *)
        feeder_running := TRUE; (* Start both feeder units and establish winding tension *)

        IF feeder_running AND NOT stop_machine THEN
            next_state := 4; (* Proceed to activate horizontal cutter *)
        ELSIF stop_machine THEN
            next_state := 6; (* Abort startup, begin shutdown *)
        ELSE
            next_state := 3; (* Wait for feeders to be confirmed running *)
        END_IF;

    4: (* Startup - Activate Horizontal Cutter *)
        cutter_running := TRUE; (* Activate the horizontal cutter *)

        IF cutter_running AND NOT stop_machine THEN
            next_state := 5; (* Proceed to final ready state (vertical cutter implied active) *)
        ELSIF stop_machine THEN
            next_state := 6; (* Abort startup, begin shutdown *)
        ELSE
            next_state := 4; (* Wait for cutter to be confirmed active *)
        END_IF;

    5: (* Startup - Ready State (Vertical Cutter active) *)
        (* Both cutters are active, machine is fully operational *)
        machine_ready := TRUE;
        startup_complete := TRUE;
        shutdown_complete := FALSE;

        IF stop_machine THEN
            next_state := 6; (* Begin normal shutdown sequence *)
        ELSE
            next_state := 5; (* Remain in ready state *)
        END_IF;

    6: (* Shutdown - Stop Both Cutters *)
        cutter_running := FALSE; (* Deactivate both horizontal and vertical cutters *)
        machine_ready := FALSE;  (* Machine is no longer ready for operation *)

        IF NOT cutter_running THEN
            next_state := 7; (* Proceed to stop feeders *)
        ELSE
            next_state := 6; (* Wait for cutters to be confirmed stopped *)
        END_IF;

    7: (* Shutdown - Stop Feeders *)
        feeder_running := FALSE; (* Stop both feeder units *)

        IF NOT feeder_running THEN
            next_state := 8; (* Proceed to deactivate heating *)
        ELSE
            next_state := 7; (* Wait for feeders to be confirmed stopped *)
        END_IF;

    8: (* Shutdown - Deactivate Heating Stations *)
        heating_running := FALSE; (* Deactivate all 8 heating stations *)

        IF NOT heating_running THEN
            next_state := 9; (* Proceed to final shutdown step *)
        ELSE
            next_state := 8; (* Wait for heating to be confirmed off *)
        END_IF;

    9: (* Shutdown - Deactivate Cooling Stations and Complete *)
        cooling_running := FALSE; (* Deactivate all 8 cooling stations *)
        shutdown_complete := TRUE;
        startup_complete := FALSE;

        IF NOT cooling_running THEN
            next_state := 0; (* Return to Idle state *)
        ELSE
            next_state := 9; (* Wait for cooling to be confirmed off *)
        END_IF;
END_CASE;

(* State Transition - Update current state for next execution cycle *)
current_state := next_state;

END_FUNCTION_BLOCK

(* ---- med_54.st ---- *)
FUNCTION_BLOCK FeedForwardControl
VAR_INPUT
    FlowRate1 : REAL; (* Input flow rate of reactant 1 *)
    FlowRate2 : REAL; (* Input flow rate of reactant 2 *)
    MixRatio  : REAL; (* Desired mixing ratio (Reactant1:Reactant2) *)
END_VAR

VAR_OUTPUT
    OutFlowRate1 : REAL; (* Output flow rate for reactant 1 *)
    OutFlowRate2 : REAL; (* Output flow rate for reactant 2 *)
END_VAR

VAR
    MixedFlowRate    : REAL; (* Total mixed flow rate *)
    ClampedFlowRate1 : REAL; (* Clamped input flow rate 1 *)
    ClampedFlowRate2 : REAL; (* Clamped input flow rate 2 *)
    RatioFactor1     : REAL; (* Ratio factor for reactant 1 *)
    RatioFactor2     : REAL; (* Ratio factor for reactant 2 *)
    PreliminaryOut1  : REAL; (* Preliminary output flow rate 1 *)
    PreliminaryOut2  : REAL; (* Preliminary output flow rate 2 *)
END_VAR

(* --- INPUT VALIDATION & CLAMPING --- *)
(* Ensure input flow rates are within the valid operating range [0, 100] *)
ClampedFlowRate1 := LIMIT(0.0, FlowRate1, 100.0);
ClampedFlowRate2 := LIMIT(0.0, FlowRate2, 100.0);

(* --- TOTAL FLOW CALCULATION --- *)
MixedFlowRate := ClampedFlowRate1 + ClampedFlowRate2;

(* --- OUTPUT CALCULATION WITH RATIO HANDLING --- *)
(* Check for invalid mixing ratio to prevent division by zero *)
IF MixRatio <> 0.0 THEN
    (* Calculate ratio factors based on MixRatio = Reactant1:Reactant2 *)
    RatioFactor1 := MixRatio / (MixRatio + 1.0);
    RatioFactor2 := 1.0 / (MixRatio + 1.0);

    (* Calculate preliminary output flow rates *)
    PreliminaryOut1 := MixedFlowRate * RatioFactor1;
    PreliminaryOut2 := MixedFlowRate * RatioFactor2;
ELSE
    (* Invalid mixing ratio: fallback to equal distribution *)
    PreliminaryOut1 := MixedFlowRate * 0.5;
    PreliminaryOut2 := MixedFlowRate * 0.5;
END_IF;

(* --- OUTPUT CLAMPING --- *)
(* Ensure final output flow rates are within the valid operating range [0, 100] *)
OutFlowRate1 := LIMIT(0.0, PreliminaryOut1, 100.0);
OutFlowRate2 := LIMIT(0.0, PreliminaryOut2, 100.0);

END_FUNCTION_BLOCK

(* ---- med_55.st ---- *)
FUNCTION_BLOCK StateMachineControl
VAR_INPUT
    request : BOOL;
    done : BOOL;
END_VAR

VAR_OUTPUT
    listen : BOOL;
END_VAR

VAR
    state : INT := 0; (* 0 = Idle, 1 = Processing *)
END_VAR

(* State Machine Logic *)
CASE state OF
    0: (* Idle State *)
        listen := TRUE;

        (* Transition to Processing when request is TRUE *)
        IF request THEN
            state := 1;
            listen := FALSE;
        END_IF;

    1: (* Processing State *)
        listen := FALSE;

        (* Transition to Idle when done is TRUE *)
        IF done THEN
            state := 0;
        END_IF;

    ELSE
        (* Fallback to Idle state for safety *)
        state := 0;
        listen := TRUE;
END_CASE;

END_FUNCTION_BLOCK

(* ---- med_56.st ---- *)
FUNCTION_BLOCK FB_SimpleRepeat
VAR_INPUT
    INPUT_VAR1 : INT := 2;
    INPUT_COUNTER : INT := 4;
END_VAR

VAR_OUTPUT
    OUTPUT_VAR1 : INT;
END_VAR

VAR
    COUNTER : INT;
END_VAR

(* Initialize output with input value *)
OUTPUT_VAR1 := INPUT_VAR1;

(* Use local counter to preserve original input parameter *)
COUNTER := INPUT_COUNTER;

(* Execute multiplication loop at least once *)
REPEAT
    OUTPUT_VAR1 := OUTPUT_VAR1 * 2;
    COUNTER := COUNTER - 1;
UNTIL COUNTER <= 0
END_REPEAT;

END_FUNCTION_BLOCK

(* ---- med_57.st ---- *)
(*
    FUNCTION_BLOCK: FB_CourseDifferenceControl
    PURPOSE: Computes the normalized angular difference between two integer inputs (in tenths of a degree).
    LOGIC:
        - If KOMPASS_GRAD < 0, KURS_DIFF is forced to 0 (error handling).
        - Otherwise, calculates KURS - KOMPASS_GRAD.
        - Normalizes the result to the range (-1800, 1800] by adding/subtracting 3600 as needed.
    VALIDATION:
        - Ensures output is always within [-1800, 1800] for valid inputs.
        - Handles negative compass input as a special error case.
*)

TYPE
    ST_CourseDifferenceData :
    STRUCT
        KOMPASS_GRAD : INT;
        KURS : INT;
        KURS_DIFF : INT;
        Status : INT; (* Use constants: INVALID_NEGATIVE, OVERFLOW_POSITIVE, OVERFLOW_NEGATIVE, VALID *)
    END_STRUCT;
END_TYPE

TYPE
    ARY_CourseDifferenceBuffer : ARRAY[0..9] OF ST_CourseDifferenceData;
END_TYPE

FUNCTION_BLOCK FB_CourseDifferenceControl
VAR_INPUT
    KOMPASS_GRAD : INT;
    KURS : INT;
END_VAR
VAR_OUTPUT
    KURS_DIFF : INT;
END_VAR
VAR
    iDiff : INT;
END_VAR

// Primary logic: Check for invalid compass input
IF KOMPASS_GRAD < 0 THEN
    KURS_DIFF := 0;
ELSE
    // Calculate raw difference
    iDiff := KURS - KOMPASS_GRAD;

    // Normalize the difference to the range (-1800, 1800]
    // Using IF statements is more efficient and deterministic than WHILE loops for this specific wrap.
    IF iDiff > 1800 THEN
        iDiff := iDiff - 3600;
    ELSIF iDiff <= -1800 THEN
        iDiff := iDiff + 3600;
    END_IF;

    KURS_DIFF := iDiff;
END_IF;

END_FUNCTION_BLOCK

(*
    MAIN PROGRAM: Example integration and data handling.
    NOTE: This program is provided for context and integration demonstration.
    The constants for the Status field (e.g., VALID) should be defined in a global configuration.
*)
PROGRAM MAIN
VAR
    fbCourseDiff : FB_CourseDifferenceControl;
    g_CourseDifferenceControlData : ST_CourseDifferenceData;
    g_CourseDifferenceBuffer : ARY_CourseDifferenceBuffer;
    nBufferIndex : INT := 0;
    // Example status constants (should be defined in a global constants list)
    INVALID_NEGATIVE : INT := 1;
    OVERFLOW_POSITIVE : INT := 2;
    OVERFLOW_NEGATIVE : INT := 3;
    VALID : INT := 0;
END_VAR

// Call the function block with data from the structure
fbCourseDiff(
    KOMPASS_GRAD := g_CourseDifferenceControlData.KOMPASS_GRAD,
    KURS := g_CourseDifferenceControlData.KURS
);
g_CourseDifferenceControlData.KURS_DIFF := fbCourseDiff.KURS_DIFF;

// Determine the status of the calculation based on inputs and result
IF g_CourseDifferenceControlData.KOMPASS_GRAD < 0 THEN
    g_CourseDifferenceControlData.Status := INVALID_NEGATIVE;
ELSIF fbCourseDiff.KURS_DIFF > 1800 THEN
    g_CourseDifferenceControlData.Status := OVERFLOW_POSITIVE;
ELSIF fbCourseDiff.KURS_DIFF < -1800 THEN
    g_CourseDifferenceControlData.Status := OVERFLOW_NEGATIVE;
ELSE
    g_CourseDifferenceControlData.Status := VALID;
END_IF;

// Buffer the result (cyclic buffer of size 10)
IF nBufferIndex >= 0 AND nBufferIndex < 10 THEN
    g_CourseDifferenceBuffer[nBufferIndex] := g_CourseDifferenceControlData;
    nBufferIndex := nBufferIndex + 1;
    IF nBufferIndex >= 10 THEN
        nBufferIndex := 0;
    END_IF;
END_IF;

END_PROGRAM

(* ---- med_58.st ---- *)
FUNCTION_BLOCK FB_ThresholdAccumulator
VAR_INPUT
    i : INT;
END_VAR

VAR_OUTPUT
    o : INT;
END_VAR

VAR
    s1 : INT;
END_VAR

(* Initialize intermediate accumulator *)
s1 := 0;

(* Process positive input *)
IF i > 0 THEN
    s1 := s1 + i;
END_IF;

(* Apply special threshold condition *)
IF s1 = 42 THEN
    s1 := s1 + 8000;
END_IF;

(* Determine final output with non-negative constraint *)
IF s1 < 0 THEN
    o := 0;
ELSE
    o := s1;
END_IF;

END_FUNCTION_BLOCK

(* ---- med_59.st ---- *)
FUNCTION_BLOCK FB_ConditionalSelectAndAggregate
VAR_INPUT
    Z : INT;
END_VAR
VAR
    A_X : INT := 42;
    A_Y : INT := 333;
END_VAR
VAR_OUTPUT
    NEW_Z : INT;
END_VAR

IF A_X > Z THEN
    NEW_Z := A_Y;
ELSE
    NEW_Z := Z;
END_IF;
NEW_Z := NEW_Z + A_X + A_Y;

END_FUNCTION_BLOCK

(* ---- med_60.st ---- *)
(*
FUNCTION_BLOCK: FB_RequestHandler
DESCRIPTION: Implements a state machine for request handling with listening mode control.
INPUTS:
    request : BOOL - Indicates if a request has been made
    done    : BOOL - Indicates if processing is completed
OUTPUTS:
    listen  : BOOL - Indicates whether the system is in listening mode
BEHAVIOR:
    State 0 (Idle):
        - listen = TRUE
        - If request = TRUE: Transition to State 1, set listen = FALSE
    State 1 (Processing):
        - listen = FALSE
        - If done = TRUE: Transition to State 0, set listen = TRUE
*)

FUNCTION_BLOCK FB_RequestHandler
VAR_INPUT
    request : BOOL;
    done    : BOOL;
END_VAR

VAR_OUTPUT
    listen : BOOL;
END_VAR

VAR
    state : INT := 0;
END_VAR

(* Main state machine logic *)
CASE state OF
    0: (* State 0: Idle/Listening *)
        listen := TRUE;

        IF request THEN
            listen := FALSE;
            state := 1;
        END_IF;

    1: (* State 1: Processing/Not Listening *)
        listen := FALSE;

        IF done THEN
            listen := TRUE;
            state := 0;
        END_IF;

END_CASE;

END_FUNCTION_BLOCK;

(* ---- med_61.st ---- *)
TYPE
    E_Status : (eIdle, eRunning, eDone, eError);
END_TYPE

TYPE
    ST_SumData :
    STRUCT
        maxValue : INT;
        wData : DWORD; (* Changed from WORD to DWORD to prevent overflow *)
        currentIndex : INT;
        status : E_Status;
    END_STRUCT
END_TYPE

FUNCTION_BLOCK FB_Sum
VAR_INPUT
    maxValue : INT;
    bExecute : BOOL; (* Added for stateful execution control *)
END_VAR
VAR_OUTPUT
    wData : DWORD; (* Changed from WORD to DWORD *)
    status : E_Status;
    bDone : BOOL;
    bError : BOOL;
END_VAR
VAR
    internalData : ST_SumData;
    bExecutePrev : BOOL;
END_VAR

(* Initialize on first execution or when not executing *)
IF NOT bExecute AND bExecutePrev THEN
    internalData.status := eIdle;
    internalData.wData := 0;
    internalData.currentIndex := 0;
    bDone := FALSE;
    bError := FALSE;
END_IF;

(* Main execution logic *)
CASE internalData.status OF
    eIdle:
        IF bExecute AND NOT bExecutePrev THEN
            (* Validate input *)
            IF maxValue < 0 THEN
                internalData.status := eError;
                bError := TRUE;
            ELSE
                internalData.maxValue := maxValue;
                internalData.wData := 0;
                internalData.currentIndex := 0;
                internalData.status := eRunning;
            END_IF;
        END_IF;

    eRunning:
        IF internalData.currentIndex <= internalData.maxValue THEN
            internalData.wData := internalData.wData + DWORD_TO_DWORD(internalData.currentIndex);
            internalData.currentIndex := internalData.currentIndex + 1;
        ELSE
            internalData.status := eDone;
            bDone := TRUE;
        END_IF;

    eDone:
        (* Maintain state until execution command is released *)
        IF NOT bExecute THEN
            internalData.status := eIdle;
            bDone := FALSE;
        END_IF;

    eError:
        (* Maintain error state until execution command is released *)
        IF NOT bExecute THEN
            internalData.status := eIdle;
            bError := FALSE;
        END_IF;
END_CASE;

(* Update outputs *)
wData := internalData.wData;
status := internalData.status;

(* Store previous execute state for edge detection *)
bExecutePrev := bExecute;

END_FUNCTION_BLOCK;

(* ---- med_62.st ---- *)
(*
FUNCTION_BLOCK: FB_PedestrianTrafficLight
DESCRIPTION: Pedestrian traffic light control system with state machine logic.
INPUTS:
  - pedBtnPress: Pedestrian button press signal (rising edge detection)
OUTPUTS:
  - carLightIsGreen: Car traffic light green status
  - pedLightIsGreen: Pedestrian light green status
  - TimeCounter: Current timer value for state transitions
STATES:
  1: IDLE - Car green, pedestrian red, waiting for button press
  2: CAR_RED - Car red, pedestrian red, counting to pedestrian green
  3: PED_GREEN - Car red, pedestrian green, counting to pedestrian red
  4: PED_RED - Car red, pedestrian red, counting to car green
*)

FUNCTION_BLOCK FB_PedestrianTrafficLight
VAR_INPUT
    pedBtnPress : BOOL; (* Pedestrian button input *)
END_VAR

VAR_OUTPUT
    carLightIsGreen : BOOL; (* Car light status *)
    pedLightIsGreen : BOOL; (* Pedestrian light status *)
    TimeCounter : INT; (* Current counter value *)
END_VAR

VAR
    buttonPressedBefore : BOOL := FALSE; (* Rising edge detection *)
    currentState : INT := 1; (* Current state (1-4) *)
    nextState : INT := 1; (* Next state for transition *)
    pedBtnPressRisingEdge : BOOL; (* Rising edge detection internal *)
END_VAR

(* Rising edge detection for pedestrian button *)
pedBtnPressRisingEdge := pedBtnPress AND NOT buttonPressedBefore;
buttonPressedBefore := pedBtnPress;

(* Main state machine logic *)
CASE currentState OF
    1: (* IDLE: Car green, pedestrian red *)
        carLightIsGreen := TRUE;
        pedLightIsGreen := FALSE;
        TimeCounter := 0;

        IF pedBtnPressRisingEdge THEN
            nextState := 2;
        ELSE
            nextState := 1;
        END_IF;

    2: (* CAR_RED: Car red, pedestrian red, counting to 10 *)
        carLightIsGreen := FALSE;
        pedLightIsGreen := FALSE;
        TimeCounter := TimeCounter + 1;

        IF TimeCounter >= 10 THEN
            nextState := 3;
        ELSE
            nextState := 2;
        END_IF;

    3: (* PED_GREEN: Car red, pedestrian green, counting to 40 *)
        carLightIsGreen := FALSE;
        pedLightIsGreen := TRUE;
        TimeCounter := TimeCounter + 1;

        IF TimeCounter >= 40 THEN
            nextState := 4;
        ELSE
            nextState := 3;
        END_IF;

    4: (* PED_RED: Car red, pedestrian red, counting to 50 *)
        carLightIsGreen := FALSE;
        pedLightIsGreen := FALSE;
        TimeCounter := TimeCounter + 1;

        IF TimeCounter >= 50 THEN
            nextState := 1;
        ELSE
            nextState := 4;
        END_IF;

END_CASE;

(* State transition *)
currentState := nextState;

END_FUNCTION_BLOCK;

(* ---- med_63.st ---- *)
TYPE
    // No custom types required for this implementation
END_TYPE

FUNCTION_BLOCK Automated_Parking_Controller
VAR_INPUT
    EntryGateSensor : BOOL;     (* Sensor input for entry gate *)
    ExitGateSensor : BOOL;      (* Sensor input for exit gate *)
    CarDetected : BOOL;         (* Sensor input for car detection *)
END_VAR

VAR_OUTPUT
    ParkingSpaceNumber : INT := 0;          (* Allocated parking space number *)
    RetrievalInProgress : BOOL := FALSE;    (* Flag for car retrieval in progress *)
END_VAR

VAR
    ParkingSpaces : ARRAY[1..100] OF BOOL := [100(FALSE)];    (* Parking space status: TRUE=Occupied, FALSE=Available *)
    i : INT;                                                    (* Loop counter *)

    // Edge detection for sensor inputs
    EntryGateRisingEdge : R_TRIG;
    ExitGateRisingEdge : R_TRIG;
    CarDetectedRisingEdge : R_TRIG;

    // State management
    CurrentState : INT := 0;        (* 0=IDLE, 1=ALLOCATE_SPACE, 2=START_RETRIEVAL, 3=MOVE_CAR, 4=EXIT_GATE *)
    AllocatedSpace : INT := 0;      (* Temporary storage for allocated space number *)

    // Movement timer for retrieval simulation
    MoveCarTimer : TON;
    MoveCarComplete : BOOL := FALSE;
END_VAR

// Edge detection for sensor inputs
EntryGateRisingEdge(CLK := EntryGateSensor);
ExitGateRisingEdge(CLK := ExitGateSensor);
CarDetectedRisingEdge(CLK := CarDetected);

// Main state machine logic
CASE CurrentState OF
    0: (* IDLE State - Waiting for events *)
        IF EntryGateRisingEdge.Q AND (NOT RetrievalInProgress) THEN
            CurrentState := 1;    // Transition to ALLOCATE_SPACE
        ELSIF CarDetectedRisingEdge.Q AND (NOT RetrievalInProgress) THEN
            CurrentState := 2;    // Transition to START_RETRIEVAL
        ELSIF ExitGateRisingEdge.Q THEN
            CurrentState := 4;    // Transition to EXIT_GATE
        END_IF;

    1: (* ALLOCATE_SPACE State - Find and assign available parking space *)
        AllocatedSpace := 0;

        // Scan for first available parking space
        FOR i := 1 TO 100 DO
            IF (NOT ParkingSpaces[i]) AND (AllocatedSpace = 0) THEN
                AllocatedSpace := i;
            END_IF;
        END_FOR;

        // If space found, allocate it
        IF AllocatedSpace > 0 THEN
            ParkingSpaces[AllocatedSpace] := TRUE;
            ParkingSpaceNumber := AllocatedSpace;
        END_IF;

        CurrentState := 0;    // Return to IDLE

    2: (* START_RETRIEVAL State - Initiate car retrieval process *)
        RetrievalInProgress := TRUE;

        // Start movement timer (simulating car movement to exit)
        MoveCarTimer(IN := TRUE, PT := T#5S);
        MoveCarComplete := FALSE;

        CurrentState := 3;    // Transition to MOVE_CAR

    3: (* MOVE_CAR State - Execute car movement to exit gate *)
        MoveCarTimer(IN := TRUE, PT := T#5S);

        IF MoveCarTimer.Q THEN
            MoveCarComplete := TRUE;
        END_IF;

        // When movement is complete, free the parking space
        IF MoveCarComplete THEN
            IF (ParkingSpaceNumber >= 1) AND (ParkingSpaceNumber <= 100) THEN
                ParkingSpaces[ParkingSpaceNumber] := FALSE;
            END_IF;

            ParkingSpaceNumber := 0;
            RetrievalInProgress := FALSE;
            MoveCarComplete := FALSE;
            CurrentState := 0;    // Return to IDLE
        END_IF;

    4: (* EXIT_GATE State - Handle car exiting through exit gate *)
        // Free the parking space if it's currently allocated
        IF (ParkingSpaceNumber >= 1) AND (ParkingSpaceNumber <= 100) THEN
            ParkingSpaces[ParkingSpaceNumber] := FALSE;
        END_IF;

        ParkingSpaceNumber := 0;
        CurrentState := 0;    // Return to IDLE

END_CASE;

END_FUNCTION_BLOCK

FUNCTION MoveCarToExitGate : BOOL
VAR_INPUT
    SpaceNumber : INT;
END_VAR
VAR
    MovementTimer : TON;
END_VAR

// This function simulates the car movement process
// In a real system, this would interface with physical actuators
MovementTimer(IN := TRUE, PT := T#5S);

IF MovementTimer.Q THEN
    MoveCarToExitGate := TRUE;    // Movement completed
ELSE
    MoveCarToExitGate := FALSE;   // Movement in progress
END_IF;

END_FUNCTION

(* ---- med_64.st ---- *)
(* ============================================================================
   Bakery Oven Control System
   FUNCTION_BLOCK: BakeryOvenControl
   Description: Implements temperature and humidity regulation with deadband
                control and a baking timer. Ensures safe, mutually exclusive
                operation of opposing control elements.
   Author: Senior PLC Commissioning Engineer
   IEC 61131-3 Compliant
============================================================================ *)

FUNCTION_BLOCK BakeryOvenControl
VAR_INPUT
    TemperatureSensor : REAL;     (* Current oven temperature measurement (°C) *)
    HumiditySensor    : REAL;     (* Current oven humidity measurement (%RH) *)
END_VAR

VAR_OUTPUT
    HeatingElement    : BOOL;     (* Control output for heating element *)
    CoolingElement    : BOOL;     (* Control output for cooling element *)
    HumidityControl   : BOOL;     (* Control output for humidification system *)
    DehumidityControl : BOOL;     (* Control output for dehumidification system *)
    TimerRemaining    : TIME;     (* Remaining baking time for display/feedback *)
    OvenActive        : BOOL;     (* Status: TRUE when oven is on and timer > 0 *)
END_VAR

VAR
    (* Process Setpoints - Initialized when oven is off *)
    TemperatureSetpoint : REAL := 180.0;   (* Desired oven temperature (°C) *)
    HumiditySetpoint    : REAL := 60.0;    (* Desired oven humidity (%RH) *)
    BakingTimeSet       : TIME := T#30m;   (* Total baking duration *)

    (* Control Parameters *)
    TemperatureThreshold : REAL := 2.0;    (* Deadband for temperature control (°C) *)
    HumidityThreshold    : REAL := 5.0;    (* Deadband for humidity control (%RH) *)

    (* Internal State Variables *)
    OvenStatus      : BOOL := FALSE;       (* Master enable: TRUE=On, FALSE=Off *)
    TimerActive     : BOOL := FALSE;       (* Timer is currently counting down *)
    TimerOneSec     : TON;                 (* One-second interval timer *)

    (* Calculated Bounds for Control *)
    TempLowerBound  : REAL;
    TempUpperBound  : REAL;
    HumidLowerBound : REAL;
    HumidUpperBound : REAL;

    (* Internal Timer Variable *)
    internalTimerRemaining : TIME := T#0s;
END_VAR

(* ============================================================================
   Initialization and Timer Management
   - Setpoints can be configured when oven is off
   - Timer decrements at 1-second intervals when active
============================================================================ *)

(* Initialize setpoints and reset outputs when oven is turned off *)
IF NOT OvenStatus THEN
    (* Reset all control outputs *)
    HeatingElement    := FALSE;
    CoolingElement    := FALSE;
    HumidityControl   := FALSE;
    DehumidityControl := FALSE;

    (* Reset timer state *)
    TimerActive := FALSE;
    internalTimerRemaining := BakingTimeSet;
    TimerOneSec(IN:=FALSE, PT:=T#1s);

    (* Setpoints can be modified here when oven is off *)
    (* Note: In a real application, these would typically be set via HMI or recipe *)
ELSE
    (* Start timer when oven is turned on *)
    IF NOT TimerActive THEN
        TimerActive := TRUE;
        internalTimerRemaining := BakingTimeSet;
    END_IF;
END_IF;

(* One-second timer for decrementing baking time *)
TimerOneSec(IN:=TimerActive AND (internalTimerRemaining > T#0s), PT:=T#1s);

(* Decrement timer at one-second intervals *)
IF TimerOneSec.Q THEN
    IF internalTimerRemaining >= T#1s THEN
        internalTimerRemaining := internalTimerRemaining - T#1s;
    ELSE
        internalTimerRemaining := T#0s;
    END_IF;
    TimerOneSec(IN:=FALSE);  (* Reset timer for next interval *)
END_IF;

(* Stop timer and deactivate oven when time reaches zero *)
IF internalTimerRemaining = T#0s THEN
    TimerActive := FALSE;
    OvenStatus := FALSE;
END_IF;

(* Update output variable for remaining time *)
TimerRemaining := internalTimerRemaining;

(* Oven is considered active only when both enabled and timer is running *)
OvenActive := OvenStatus AND TimerActive AND (internalTimerRemaining > T#0s);

(* ============================================================================
   Safety Validation and Bound Calculation
   - Ensure thresholds are positive to prevent inverted control logic
   - Calculate control bounds with validated thresholds
============================================================================ *)

(* Validate thresholds are positive - use absolute value as safety measure *)
TemperatureThreshold := ABS(TemperatureThreshold);
HumidityThreshold := ABS(HumidityThreshold);

(* Ensure minimum threshold values to prevent excessive cycling *)
IF TemperatureThreshold < 0.1 THEN
    TemperatureThreshold := 0.1;
END_IF;

IF HumidityThreshold < 0.5 THEN
    HumidityThreshold := 0.5;
END_IF;

(* Calculate control bounds *)
TempLowerBound  := TemperatureSetpoint - TemperatureThreshold;
TempUpperBound  := TemperatureSetpoint + TemperatureThreshold;
HumidLowerBound := HumiditySetpoint - HumidityThreshold;
HumidUpperBound := HumiditySetpoint + HumidityThreshold;

(* ============================================================================
   Temperature Control Logic
   - Heating activates when temperature < lower bound
   - Cooling activates when temperature > upper bound
   - Explicit mutual exclusion between heating and cooling
   - Both off when within deadband
============================================================================ *)

IF OvenActive THEN
    (* Temperature Control with Explicit Mutual Exclusion *)
    IF TemperatureSensor < TempLowerBound THEN
        (* Temperature too low - activate heating *)
        HeatingElement := TRUE;
        CoolingElement := FALSE;
    ELSIF TemperatureSensor > TempUpperBound THEN
        (* Temperature too high - activate cooling *)
        HeatingElement := FALSE;
        CoolingElement := TRUE;
    ELSE
        (* Temperature within acceptable range *)
        HeatingElement := FALSE;
        CoolingElement := FALSE;
    END_IF;

    (* Humidity Control with Explicit Mutual Exclusion *)
    IF HumiditySensor < HumidLowerBound THEN
        (* Humidity too low - activate humidification *)
        HumidityControl := TRUE;
        DehumidityControl := FALSE;
    ELSIF HumiditySensor > HumidUpperBound THEN
        (* Humidity too high - activate dehumidification *)
        HumidityControl := FALSE;
        DehumidityControl := TRUE;
    ELSE
        (* Humidity within acceptable range *)
        HumidityControl := FALSE;
        DehumidityControl := FALSE;
    END_IF;
ELSE
    (* Oven not active - force all outputs off *)
    HeatingElement    := FALSE;
    CoolingElement    := FALSE;
    HumidityControl   := FALSE;
    DehumidityControl := FALSE;
END_IF;

(* ============================================================================
   Final Safety Interlock
   - Redundant protection against simultaneous activation
   - Ensures outputs are forced off when oven is not active
============================================================================ *)

(* Final mutual exclusion check - redundant safety *)
IF HeatingElement AND CoolingElement THEN
    HeatingElement := FALSE;
    CoolingElement := FALSE;
END_IF;

IF HumidityControl AND DehumidityControl THEN
    HumidityControl := FALSE;
    DehumidityControl := FALSE;
END_IF;

(* Master disable - final override *)
IF NOT OvenActive THEN
    HeatingElement    := FALSE;
    CoolingElement    := FALSE;
    HumidityControl   := FALSE;
    DehumidityControl := FALSE;
END_IF;

END_FUNCTION_BLOCK;

(* ---- med_65.st ---- *)
FUNCTION_BLOCK TheaterControl
VAR_INPUT
    StartButton : BOOL; (* Input for starting a performance *)
    StopButton : BOOL; (* Input for stopping a performance *)
    SceneNumber : INT; (* Input for selecting the scene or act *)
END_VAR

VAR_OUTPUT
    LightingControl : BOOL; (* Output for controlling lighting *)
    SoundControl : BOOL; (* Output for controlling sound *)
    PerformanceInProgress : BOOL; (* Indicator for an ongoing performance *)
END_VAR

VAR
    bStartRisingEdge : BOOL; (* Detects rising edge of StartButton *)
    bPrevStartState : BOOL; (* Previous state for edge detection *)
END_VAR

(* Rising edge detection for StartButton *)
bStartRisingEdge := StartButton AND NOT bPrevStartState;
bPrevStartState := StartButton;

(* Main control logic with StopButton as highest priority *)
IF StopButton THEN
    (* Immediate halt: override all other inputs *)
    PerformanceInProgress := FALSE;
    LightingControl := FALSE;
    SoundControl := FALSE;
ELSIF bStartRisingEdge AND NOT PerformanceInProgress THEN
    (* Start attempt when not already in progress *)
    IF (SceneNumber >= 1) AND (SceneNumber <= 3) THEN
        (* Valid scene: activate performance *)
        PerformanceInProgress := TRUE;
        LightingControl := TRUE;
        SoundControl := TRUE;
    ELSE
        (* Invalid scene: ensure all outputs are FALSE *)
        PerformanceInProgress := FALSE;
        LightingControl := FALSE;
        SoundControl := FALSE;
    END_IF;
END_IF;

(* Note: Once started, outputs remain TRUE until StopButton is pressed.
   The PerformanceInProgress state persists between cycles,
   preventing re-triggering while active. *)
END_FUNCTION_BLOCK;

(* ---- med_66.st ---- *)
(*
    Elevator Control System Function Block
    Author: Senior PLC Commissioning Engineer
    Description: Controls elevator movement and door operations based on position requests
    Compliance: IEC 61131-3 Structured Text
*)

FUNCTION_BLOCK ElevatorControl
VAR_INPUT
    CurrentPos : INT;           (* Current floor position *)
    RequestedPos : INT;         (* Target floor position *)
    ButtonPressed : BOOL;       (* Button press trigger *)
END_VAR

VAR_OUTPUT
    MotorMovingUp : BOOL;       (* Elevator moving upward *)
    MotorMovingDown : BOOL;     (* Elevator moving downward *)
    DoorIsOpen : BOOL;          (* Door open status *)
END_VAR

VAR
    (* State machine enumeration *)
    State : (IDLE, MOVING_UP, MOVING_DOWN);

    (* Edge detection for button press *)
    PrevButtonPressed : BOOL := FALSE;

    (* Internal target storage for dynamic updates *)
    ActiveTarget : INT := 0;

    (* Safety flag to prevent simultaneous motor activation *)
    MotorActive : BOOL := FALSE;
END_VAR

(* Main state machine logic *)
CASE State OF
    IDLE:
        (* Stationary state - door open, motors off *)
        MotorMovingUp := FALSE;
        MotorMovingDown := FALSE;
        DoorIsOpen := TRUE;
        MotorActive := FALSE;

        (* Check for new button press with edge detection *)
        IF ButtonPressed AND NOT PrevButtonPressed THEN
            (* Store the requested position for dynamic updates *)
            ActiveTarget := RequestedPos;

            (* Determine movement direction *)
            IF ActiveTarget > CurrentPos THEN
                State := MOVING_UP;
                DoorIsOpen := FALSE;
                MotorMovingUp := TRUE;
                MotorActive := TRUE;
            ELSIF ActiveTarget < CurrentPos THEN
                State := MOVING_DOWN;
                DoorIsOpen := FALSE;
                MotorMovingDown := TRUE;
                MotorActive := TRUE;
            ELSE
                (* Already at target floor *)
                DoorIsOpen := TRUE;
                State := IDLE;
            END_IF;
        END_IF;

        (* Monitor for dynamic target updates while idle *)
        IF RequestedPos <> ActiveTarget AND ButtonPressed AND NOT PrevButtonPressed THEN
            ActiveTarget := RequestedPos;
        END_IF;

    MOVING_UP:
        (* Elevator moving upward *)
        MotorMovingUp := TRUE;
        MotorMovingDown := FALSE;
        DoorIsOpen := FALSE;
        MotorActive := TRUE;

        (* Check for dynamic target updates during movement *)
        IF RequestedPos <> ActiveTarget THEN
            ActiveTarget := RequestedPos;

            (* Re-evaluate direction if target changes *)
            IF ActiveTarget < CurrentPos THEN
                State := MOVING_DOWN;
            ELSIF ActiveTarget = CurrentPos THEN
                State := IDLE;
            END_IF;
        END_IF;

        (* Check if target floor reached *)
        IF CurrentPos >= ActiveTarget THEN
            (* Exact position check for safety *)
            IF CurrentPos = ActiveTarget THEN
                State := IDLE;
                MotorMovingUp := FALSE;
                DoorIsOpen := TRUE;
                MotorActive := FALSE;
            END_IF;
        END_IF;

    MOVING_DOWN:
        (* Elevator moving downward *)
        MotorMovingUp := FALSE;
        MotorMovingDown := TRUE;
        DoorIsOpen := FALSE;
        MotorActive := TRUE;

        (* Check for dynamic target updates during movement *)
        IF RequestedPos <> ActiveTarget THEN
            ActiveTarget := RequestedPos;

            (* Re-evaluate direction if target changes *)
            IF ActiveTarget > CurrentPos THEN
                State := MOVING_UP;
            ELSIF ActiveTarget = CurrentPos THEN
                State := IDLE;
            END_IF;
        END_IF;

        (* Check if target floor reached *)
        IF CurrentPos <= ActiveTarget THEN
            (* Exact position check for safety *)
            IF CurrentPos = ActiveTarget THEN
                State := IDLE;
                MotorMovingDown := FALSE;
                DoorIsOpen := TRUE;
                MotorActive := FALSE;
            END_IF;
        END_IF;

END_CASE;

(* Update button press history for edge detection *)
PrevButtonPressed := ButtonPressed;

(* Safety interlock: Ensure motors are never active simultaneously *)
IF MotorMovingUp AND MotorMovingDown THEN
    MotorMovingUp := FALSE;
    MotorMovingDown := FALSE;
    MotorActive := FALSE;
    State := IDLE;
END_IF;

END_FUNCTION_BLOCK

(* ---- med_67.st ---- *)
TYPE
    E_CalculationStatus : (eStatus_InvalidInput, eStatus_ValidInput, eStatus_OverflowPrevented);
END_TYPE

FUNCTION_BLOCK FB_FactorialCalculator
VAR_INPUT
    X : INT;
END_VAR

VAR_OUTPUT
    FactorialResult : INT;
    FactorialGoodResult : INT;
    eStatus : E_CalculationStatus;
END_VAR

VAR
    nTempGoodResult : INT;
END_VAR

(* Initialize outputs *)
FactorialGoodResult := 0;
FactorialResult := 1;
eStatus := eStatus_InvalidInput;

(* Check input range *)
IF (X >= -3) AND (X <= 3) THEN
    (* Calculate FactorialGoodResult as X⁴ *)
    nTempGoodResult := X * X * X * X;
    FactorialGoodResult := nTempGoodResult;

    (* Calculate FactorialResult based on FactorialGoodResult *)
    IF nTempGoodResult > 1 THEN
        FactorialResult := nTempGoodResult * (nTempGoodResult - 1);
    ELSE
        FactorialResult := nTempGoodResult;
    END_IF;

    eStatus := eStatus_ValidInput;
ELSE
    (* Handle out-of-range input to prevent overflow *)
    FactorialGoodResult := 0;
    FactorialResult := 1;
    eStatus := eStatus_OverflowPrevented;
END_IF;

END_FUNCTION_BLOCK;

(* ---- med_68.st ---- *)
FUNCTION_BLOCK FB_SignalControl
VAR_INPUT
    Int1 : BOOL;
    Int2 : BOOL;
    Int3 : BOOL;
    Int4 : BOOL;
    Int5 : BOOL;
    Int6 : BOOL;
    Int7 : BOOL;
    Int8 : BOOL;
    IntAn1 : UINT;
    IntAn2 : UINT;
    IntAn3 : UINT;
    IntAn4 : UINT;
    IntAn5 : UINT;
    IntAn6 : UINT;
    IntAn7 : UINT;
    IntAn8 : UINT;
    Marca2 : BOOL;
END_VAR

VAR_OUTPUT
    Out1 : BOOL;
    Out2 : BOOL;
    Out3 : BOOL;
    Out4 : BOOL;
    Out5 : BOOL;
    Out6 : BOOL;
    Out7 : BOOL;
    Out8 : BOOL;
    OutAn1 : UINT;
    OutAn2 : UINT;
    OutAn3 : UINT;
    OutAn4 : UINT;
    OutAn5 : UINT;
    OutAn6 : UINT;
    OutAn7 : UINT;
    OutAn8 : UINT;
END_VAR

VAR
    Marca1 : BOOL;
END_VAR

// Logic Implementation

// 1. Latch Logic for Out1 using Marca1 and Marca2
// Marca1 condition: Set when Marca2 is FALSE AND (Marca1 is TRUE OR Out1 is FALSE) AND Int1 is TRUE
Marca1 := (NOT Marca2) AND (Marca1 OR NOT Out1) AND Int1;

// Marca2 condition: Set when Marca1 is FALSE AND (Marca2 is TRUE OR Out1 is TRUE) AND Int1 is TRUE
// Note: Marca2 is an input, so we don't assign to it. The description suggests it should be internal,
// but the interface defines it as input. We'll use the input value directly.

// Out1 latch condition: Set when Marca2 is FALSE AND (Marca1 is TRUE OR Out1 is TRUE)
Out1 := (NOT Marca2) AND (Marca1 OR Out1);

// 2. Direct Boolean Pass-Through
Out2 := Int2;
Out3 := Int3;
Out4 := Int4;

// 3. Direct Analog Pass-Through
OutAn1 := IntAn1;
OutAn2 := IntAn2;
OutAn3 := IntAn3;
OutAn4 := IntAn4;
OutAn5 := IntAn5;
OutAn6 := IntAn6;
OutAn7 := IntAn7;
OutAn8 := IntAn8;

// 4. Conditional Output Logic for Out5 to Out8
Out5 := (IntAn5 > 1000) AND NOT Int5;
Out6 := (IntAn6 > 1000) AND NOT Int6;
Out7 := (IntAn7 > 1000) AND NOT Int7;
Out8 := (IntAn8 > 1000) AND NOT Int8;

END_FUNCTION_BLOCK;
